SPLINE
SPL {X  -159.990, Y  +457.098, Z    +0.000, E1   +61.912, E3 +184875.364}
SPL {X  -159.990, Y  +442.075, Z    +0.000, E1   +62.596, E3 +184887.140}
SPL {X  -159.990, Y  +430.868, Z    +0.000, E1   +63.135, E3 +184895.393}
SPL {X  -159.990, Y  +416.857, Z    +0.000, E1   +63.835, E3 +184905.060}
SPL {X  -159.990, Y  +402.942, Z    +0.000, E1   +64.377, E3 +184915.289}
SPL {X  -159.990, Y  +382.745, Z    +0.000, E1   +65.209, E3 +184929.203}
SPL {X  -158.929, Y  +364.101, Z    +0.000, E1   +65.981, E3 +184940.958}
SPL {X  -156.693, Y  +350.188, Z    +0.000, E1   +66.345, E3 +184951.082}
SPL {X  -154.578, Y  +341.238, Z    +0.000, E1   +66.113, E3 +184960.840}
SPL {X  -151.958, Y  +332.444, Z    +0.000, E1   +65.791, E3 +184971.400}
SPL {X  -148.012, Y  +321.760, Z    +0.000, E1   +65.212, E3 +184985.033}
SPL {X  -145.172, Y  +315.256, Z    +0.000, E1   +64.753, E3 +184993.738}
SPL {X  -142.205, Y  +309.188, Z    +0.000, E1   +64.322, E3 +185001.991}
SPL {X  -138.693, Y  +302.744, Z    +0.000, E1   +63.741, E3 +185011.048}
SPL {X  -135.977, Y  +298.197, Z    +0.000, E1   +63.280, E3 +185017.568}
SPL {X  -132.828, Y  +293.318, Z    +0.000, E1   +62.759, E3 +185024.622}
SPL {X  -129.451, Y  +288.482, Z    +0.000, E1   +62.137, E3 +185031.725}
SPL {X  -102.192, Y  +259.400, Z    +0.000, E1   +52.167, E3 +185148.272}
ENDSPLINE

SPLINE
SPL {X  -140.725, Y  +306.386, Z    +0.000, E1   +41.058, E3 +185273.166}
SPL {X  -153.851, Y  +338.606, Z    +0.000, E1   +29.149, E3 +185289.783}
SPL {X  -158.264, Y  +359.064, Z    +0.000, E1   +18.155, E3 +185294.734}
SPL {X  -159.641, Y  +371.933, Z    +0.000, E1    +9.693, E3 +185296.470}
SPL {X  -159.986, Y  +381.420, Z    +0.000, E1    +2.704, E3 +185297.035}
SPL {X  -159.990, Y  +384.527, Z    +0.000, E1    -0.013, E3 +185297.095}
SPL {X  -159.990, Y  +385.909, Z    +0.000, E1    -1.800, E3 +185297.113}
SPL {X  -159.990, Y  +389.230, Z    +0.000, E1    -6.815, E3 +185297.237}
SPL {X  -159.990, Y  +395.332, Z    +0.000, E1   -17.451, E3 +185297.720}
SPL {X  -159.990, Y  +403.857, Z    +0.000, E1   -31.979, E3 +185298.945}
SPL {X  -159.990, Y  +417.858, Z    +0.000, E1   -47.695, E3 +185302.430}
SPL {X  -159.990, Y  +475.808, Z    +0.000, E1   -64.751, E3 +185326.384}
SPL {X  -159.990, Y  +590.266, Z    +0.000, E1   -66.680, E3 +185409.501}
SPL {X  -159.990, Y  +605.903, Z    +0.000, E1   -66.635, E3 +185423.920}
SPL {X  -159.990, Y  +620.525, Z    +0.000, E1   -66.669, E3 +185437.254}
SPL {X  -159.990, Y  +638.202, Z    +0.000, E1   -66.649, E3 +185453.504}
SPL {X  -159.990, Y  +654.774, Z    +0.000, E1   -66.658, E3 +185468.673}
SPL {X  -159.990, Y  +671.049, Z    +0.000, E1   -66.648, E3 +185483.604}
SPL {X  -159.584, Y  +682.893, Z    +0.000, E1   -66.583, E3 +185494.902}
SPL {X  -158.845, Y  +690.607, Z    +0.000, E1   -66.486, E3 +185502.754}
SPL {X  -157.279, Y  +700.830, Z    +0.000, E1   -66.296, E3 +185513.735}
SPL {X  -154.589, Y  +712.719, Z    +0.000, E1   -65.941, E3 +185527.378}
SPL {X  -151.974, Y  +721.507, Z    +0.000, E1   -65.548, E3 +185538.131}
SPL {X  -149.510, Y  +728.452, Z    +0.000, E1   -65.197, E3 +185546.973}
SPL {X  -146.809, Y  +735.092, Z    +0.000, E1   -64.789, E3 +185555.720}
SPL {X  -143.550, Y  +742.141, Z    +0.000, E1   -64.312, E3 +185565.239}
SPL {X  -140.309, Y  +748.378, Z    +0.000, E1   -63.779, E3 +185573.972}
SPL {X  -136.621, Y  +754.755, Z    +0.000, E1   -63.190, E3 +185583.089}
SPL {X  -133.172, Y  +760.168, Z    +0.000, E1   -62.565, E3 +185591.010}
SPL {X  -130.070, Y  +764.659, Z    +0.000, E1   -62.024, E3 +185597.606}
SPL {X  -103.420, Y  +793.570, Z    +0.000, E1   -51.337, E3 +185727.505}
ENDSPLINE

SPLINE
SPL {X  -141.359, Y  +746.429, Z    +0.000, E1   -41.207, E3 +185845.719}
SPL {X  -153.791, Y  +715.605, Z    +0.000, E1   -29.700, E3 +185860.488}
SPL {X  -157.923, Y  +697.131, Z    +0.000, E1   -19.758, E3 +185865.020}
SPL {X  -159.426, Y  +684.927, Z    +0.000, E1   -11.876, E3 +185866.749}
SPL {X  -159.929, Y  +675.915, Z    +0.000, E1    -5.290, E3 +185867.459}
SPL {X  -159.990, Y  +669.794, Z    +0.000, E1    -0.371, E3 +185867.633}
SPL {X  -159.990, Y  +668.338, Z    +0.000, E1    +1.468, E3 +185867.649}
SPL {X  -159.990, Y  +664.217, Z    +0.000, E1    +7.944, E3 +185867.802}
SPL {X  -159.990, Y  +657.963, Z    +0.000, E1   +19.417, E3 +185868.298}
SPL {X  -159.990, Y  +649.570, Z    +0.000, E1   +33.681, E3 +185869.522}
SPL {X  -159.990, Y  +636.314, Z    +0.000, E1   +48.490, E3 +185872.825}
SPL {X  -159.990, Y  +588.081, Z    +0.000, E1   +63.406, E3 +185894.007}
SPL {X  -159.990, Y  +471.514, Z    +0.000, E1   +66.231, E3 +185977.515}
SPL {X  -159.990, Y  +458.012, Z    +0.000, E1   +66.224, E3 +185990.144}
SPL {X  -159.990, Y  +445.900, Z    +0.000, E1   +66.225, E3 +186001.458}
ENDSPLINE

SPLINE
SPL {X  -159.990, Y  +465.730, Z    +0.000, E1   +61.693, E3 +186015.282}
ENDSPLINE

SPLINE
SPL {X  -159.990, Y  +446.910, Z    +0.000, E1   +62.394, E3 +186031.502}
SPL {X  -159.990, Y  +430.868, Z    +0.000, E1   +63.135, E3 +186043.542}
SPL {X  -159.990, Y  +416.857, Z    +0.000, E1   +63.835, E3 +186053.208}
SPL {X  -159.990, Y  +402.942, Z    +0.000, E1   +64.377, E3 +186063.437}
SPL {X  -159.990, Y  +382.745, Z    +0.000, E1   +65.209, E3 +186077.352}
SPL {X  -158.342, Y  +359.598, Z    +0.000, E1   +66.150, E3 +186092.056}
SPL {X  -155.453, Y  +344.669, Z    +0.000, E1   +66.270, E3 +186104.898}
SPL {X  -151.958, Y  +332.444, Z    +0.000, E1   +65.791, E3 +186119.548}
SPL {X  -148.012, Y  +321.760, Z    +0.000, E1   +65.212, E3 +186133.181}
SPL {X  -144.181, Y  +313.155, Z    +0.000, E1   +64.628, E3 +186144.691}
SPL {X  -141.300, Y  +307.460, Z    +0.000, E1   +64.150, E3 +186152.583}
SPL {X  -138.693, Y  +302.744, Z    +0.000, E1   +63.741, E3 +186159.196}
SPL {X  -135.031, Y  +296.690, Z    +0.000, E1   +63.147, E3 +186167.858}
SPL {X  -130.494, Y  +289.936, Z    +0.000, E1   +62.364, E3 +186177.696}
SPL {X  -102.192, Y  +259.400, Z    +0.000, E1   +52.167, E3 +186296.420}
ENDSPLINE

SPLINE
SPL {X  -140.725, Y  +306.386, Z    +0.000, E1   +41.058, E3 +186421.314}
SPL {X  -153.851, Y  +338.606, Z    +0.000, E1   +29.149, E3 +186437.932}
SPL {X  -158.264, Y  +359.064, Z    +0.000, E1   +18.155, E3 +186442.883}
SPL {X  -159.641, Y  +371.933, Z    +0.000, E1    +9.693, E3 +186444.618}
SPL {X  -159.986, Y  +381.420, Z    +0.000, E1    +2.704, E3 +186445.183}
SPL {X  -159.990, Y  +384.527, Z    +0.000, E1    -0.013, E3 +186445.244}
SPL {X  -159.990, Y  +386.984, Z    +0.000, E1    -3.187, E3 +186445.295}
SPL {X  -159.990, Y  +392.544, Z    +0.000, E1   -12.471, E3 +186445.608}
SPL {X  -159.990, Y  +397.827, Z    +0.000, E1   -22.184, E3 +186446.129}
SPL {X  -159.990, Y  +403.857, Z    +0.000, E1   -31.979, E3 +186447.093}
SPL {X  -159.990, Y  +417.858, Z    +0.000, E1   -47.695, E3 +186450.579}
SPL {X  -159.990, Y  +475.808, Z    +0.000, E1   -64.751, E3 +186474.532}
SPL {X  -159.990, Y  +586.159, Z    +0.000, E1   -66.648, E3 +186553.948}
SPL {X  -159.990, Y  +602.026, Z    +0.000, E1   -66.659, E3 +186568.465}
SPL {X  -159.990, Y  +620.525, Z    +0.000, E1   -66.669, E3 +186585.402}
SPL {X  -159.990, Y  +638.202, Z    +0.000, E1   -66.649, E3 +186601.652}
SPL {X  -159.990, Y  +654.774, Z    +0.000, E1   -66.658, E3 +186616.821}
SPL {X  -159.990, Y  +671.049, Z    +0.000, E1   -66.648, E3 +186631.752}
SPL {X  -159.230, Y  +687.071, Z    +0.000, E1   -66.569, E3 +186647.193}
SPL {X  -157.279, Y  +700.830, Z    +0.000, E1   -66.296, E3 +186661.883}
SPL {X  -154.589, Y  +712.719, Z    +0.000, E1   -65.941, E3 +186675.526}
SPL {X  -151.974, Y  +721.507, Z    +0.000, E1   -65.548, E3 +186686.279}
SPL {X  -149.510, Y  +728.452, Z    +0.000, E1   -65.197, E3 +186695.121}
SPL {X  -145.784, Y  +737.407, Z    +0.000, E1   -64.671, E3 +186706.912}
SPL {X  -141.166, Y  +746.792, Z    +0.000, E1   -63.950, E3 +186719.841}
SPL {X  -136.621, Y  +754.755, Z    +0.000, E1   -63.190, E3 +186731.237}
SPL {X  -133.172, Y  +760.168, Z    +0.000, E1   -62.565, E3 +186739.158}
SPL {X  -130.070, Y  +764.659, Z    +0.000, E1   -62.024, E3 +186745.754}
SPL {X  -103.420, Y  +793.570, Z    +0.000, E1   -51.337, E3 +186875.653}
ENDSPLINE

SPLINE
SPL {X  -132.256, Y  +761.529, Z    +0.000, E1   -44.935, E3 +186981.743}
SPL {X  -148.790, Y  +730.309, Z    +0.000, E1   -35.907, E3 +187003.017}
SPL {X  -157.132, Y  +701.603, Z    +0.000, E1   -22.438, E3 +187012.278}
SPL {X  -159.426, Y  +684.927, Z    +0.000, E1   -11.876, E3 +187014.897}
SPL {X  -159.929, Y  +675.915, Z    +0.000, E1    -5.290, E3 +187015.607}
SPL {X  -159.990, Y  +669.794, Z    +0.000, E1    -0.371, E3 +187015.781}
SPL {X  -159.990, Y  +668.338, Z    +0.000, E1    +1.468, E3 +187015.797}
SPL {X  -159.990, Y  +664.217, Z    +0.000, E1    +7.944, E3 +187015.950}
SPL {X  -159.990, Y  +657.963, Z    +0.000, E1   +19.417, E3 +187016.446}
SPL {X  -159.990, Y  +649.570, Z    +0.000, E1   +33.681, E3 +187017.670}
SPL {X  -159.990, Y  +636.314, Z    +0.000, E1   +48.490, E3 +187020.974}
SPL {X  -159.990, Y  +588.081, Z    +0.000, E1   +63.406, E3 +187042.155}
SPL {X  -159.990, Y  +471.514, Z    +0.000, E1   +66.231, E3 +187125.663}
SPL {X  -159.990, Y  +458.012, Z    +0.000, E1   +66.224, E3 +187138.293}
SPL {X  -159.990, Y  +445.900, Z    +0.000, E1   +66.225, E3 +187149.606}
ENDSPLINE

SPLINE
SPL {X  -159.990, Y  +465.730, Z    +0.000, E1   +61.693, E3 +187163.430}
ENDSPLINE

SPLINE
SPL {X  -159.990, Y  +452.456, Z    +0.000, E1   +62.114, E3 +187175.358}
SPL {X  -159.990, Y  +436.367, Z    +0.000, E1   +62.893, E3 +187187.618}
SPL {X  -159.990, Y  +416.857, Z    +0.000, E1   +63.835, E3 +187201.357}
SPL {X  -159.990, Y  +402.942, Z    +0.000, E1   +64.377, E3 +187211.585}
SPL {X  -159.990, Y  +382.745, Z    +0.000, E1   +65.209, E3 +187225.500}
SPL {X  -158.342, Y  +359.598, Z    +0.000, E1   +66.150, E3 +187240.204}
SPL {X  -155.453, Y  +344.669, Z    +0.000, E1   +66.270, E3 +187253.046}
SPL {X  -151.958, Y  +332.444, Z    +0.000, E1   +65.791, E3 +187267.696}
SPL {X  -148.012, Y  +321.760, Z    +0.000, E1   +65.212, E3 +187281.329}
SPL {X  -144.181, Y  +313.155, Z    +0.000, E1   +64.628, E3 +187292.839}
SPL {X  -141.300, Y  +307.460, Z    +0.000, E1   +64.150, E3 +187300.731}
SPL {X  -138.693, Y  +302.744, Z    +0.000, E1   +63.741, E3 +187307.345}
SPL {X  -135.031, Y  +296.690, Z    +0.000, E1   +63.147, E3 +187316.006}
SPL {X  -130.494, Y  +289.936, Z    +0.000, E1   +62.364, E3 +187325.844}
SPL {X  -102.192, Y  +259.400, Z    +0.000, E1   +52.167, E3 +187444.569}
ENDSPLINE

SPLINE
SPL {X  -140.725, Y  +306.386, Z    +0.000, E1   +41.058, E3 +187569.463}
SPL {X  -153.851, Y  +338.606, Z    +0.000, E1   +29.149, E3 +187586.080}
SPL {X  -157.523, Y  +354.512, Z    +0.000, E1   +20.811, E3 +187590.206}
SPL {X  -159.458, Y  +369.460, Z    +0.000, E1   +11.469, E3 +187592.495}
SPL {X  -159.986, Y  +381.420, Z    +0.000, E1    +2.704, E3 +187593.331}
SPL {X  -159.990, Y  +385.016, Z    +0.000, E1    -0.442, E3 +187593.398}
SPL {X  -159.990, Y  +389.230, Z    +0.000, E1    -6.815, E3 +187593.534}
SPL {X  -159.990, Y  +395.332, Z    +0.000, E1   -17.451, E3 +187594.016}
SPL {X  -159.990, Y  +403.857, Z    +0.000, E1   -31.979, E3 +187595.241}
SPL {X  -159.990, Y  +416.313, Z    +0.000, E1   -46.481, E3 +187598.234}
SPL {X  -159.990, Y  +425.447, Z    +0.000, E1   -52.896, E3 +187601.143}
SPL {X  -159.990, Y  +475.808, Z    +0.000, E1   -64.751, E3 +187622.680}
SPL {X  -159.990, Y  +586.159, Z    +0.000, E1   -66.648, E3 +187702.096}
SPL {X  -159.990, Y  +602.026, Z    +0.000, E1   -66.659, E3 +187716.613}
SPL {X  -159.990, Y  +615.972, Z    +0.000, E1   -66.639, E3 +187729.441}
SPL {X  -159.990, Y  +629.811, Z    +0.000, E1   -66.653, E3 +187742.093}
SPL {X  -159.990, Y  +646.024, Z    +0.000, E1   -66.650, E3 +187756.970}
SPL {X  -159.990, Y  +658.527, Z    +0.000, E1   -66.634, E3 +187768.451}
SPL {X  -159.990, Y  +671.049, Z    +0.000, E1   -66.648, E3 +187779.900}
SPL {X  -159.584, Y  +682.893, Z    +0.000, E1   -66.583, E3 +187791.198}
SPL {X  -158.332, Y  +694.472, Z    +0.000, E1   -66.450, E3 +187803.071}
SPL {X  -156.148, Y  +706.350, Z    +0.000, E1   -66.133, E3 +187816.283}
SPL {X  -154.052, Y  +714.685, Z    +0.000, E1   -65.842, E3 +187826.070}
SPL {X  -151.381, Y  +723.275, Z    +0.000, E1   -65.482, E3 +187836.617}
SPL {X  -147.622, Y  +733.180, Z    +0.000, E1   -64.943, E3 +187849.421}
SPL {X  -144.546, Y  +740.079, Z    +0.000, E1   -64.439, E3 +187858.749}
SPL {X  -142.587, Y  +744.066, Z    +0.000, E1   -64.133, E3 +187864.243}
SPL {X  -139.326, Y  +750.145, Z    +0.000, E1   -63.650, E3 +187872.736}
SPL {X  -135.791, Y  +756.103, Z    +0.000, E1   -63.018, E3 +187881.381}
SPL {X  -133.172, Y  +760.168, Z    +0.000, E1   -62.565, E3 +187887.306}
SPL {X  -130.070, Y  +764.659, Z    +0.000, E1   -62.024, E3 +187893.902}
SPL {X  -103.420, Y  +793.570, Z    +0.000, E1   -51.337, E3 +188023.802}
ENDSPLINE

SPLINE
SPL {X  -132.256, Y  +761.529, Z    +0.000, E1   -44.935, E3 +188129.891}
SPL {X  -148.790, Y  +730.309, Z    +0.000, E1   -35.907, E3 +188151.165}
SPL {X  -157.132, Y  +701.603, Z    +0.000, E1   -22.438, E3 +188160.426}
SPL {X  -159.426, Y  +684.927, Z    +0.000, E1   -11.876, E3 +188163.045}
SPL {X  -159.929, Y  +675.915, Z    +0.000, E1    -5.290, E3 +188163.755}
SPL {X  -159.990, Y  +669.794, Z    +0.000, E1    -0.371, E3 +188163.929}
SPL {X  -159.990, Y  +668.338, Z    +0.000, E1    +1.468, E3 +188163.945}
SPL {X  -159.990, Y  +665.597, Z    +0.000, E1    +5.793, E3 +188164.024}
SPL {X  -159.990, Y  +662.769, Z    +0.000, E1   +10.720, E3 +188164.175}
SPL {X  -159.990, Y  +657.963, Z    +0.000, E1   +19.417, E3 +188164.595}
SPL {X  -159.990, Y  +649.570, Z    +0.000, E1   +33.681, E3 +188165.819}
SPL {X  -159.990, Y  +636.314, Z    +0.000, E1   +48.490, E3 +188169.122}
SPL {X  -159.990, Y  +588.081, Z    +0.000, E1   +63.406, E3 +188190.303}
SPL {X  -159.990, Y  +471.514, Z    +0.000, E1   +66.231, E3 +188273.811}
SPL {X  -159.990, Y  +458.012, Z    +0.000, E1   +66.224, E3 +188286.441}
SPL {X  -159.990, Y  +445.900, Z    +0.000, E1   +66.225, E3 +188297.754}
ENDSPLINE

SPLINE
SPL {X  -159.990, Y  +465.730, Z    +0.000, E1   +61.693, E3 +188311.579}
ENDSPLINE

SPLINE
SPL {X  -159.990, Y  +446.910, Z    +0.000, E1   +62.394, E3 +188327.798}
SPL {X  -159.990, Y  +430.868, Z    +0.000, E1   +63.135, E3 +188339.838}
SPL {X  -159.990, Y  +416.857, Z    +0.000, E1   +63.835, E3 +188349.505}
SPL {X  -159.990, Y  +397.192, Z    +0.000, E1   +64.622, E3 +188363.798}
SPL {X  -159.570, Y  +370.917, Z    +0.000, E1   +65.713, E3 +188381.155}
SPL {X  -156.693, Y  +350.188, Z    +0.000, E1   +66.345, E3 +188395.527}
SPL {X  -153.533, Y  +337.508, Z    +0.000, E1   +66.008, E3 +188409.659}
SPL {X  -150.132, Y  +327.208, Z    +0.000, E1   +65.515, E3 +188422.445}
SPL {X  -146.325, Y  +317.802, Z    +0.000, E1   +64.967, E3 +188434.700}
SPL {X  -142.205, Y  +309.188, Z    +0.000, E1   +64.322, E3 +188446.436}
SPL {X  -138.693, Y  +302.744, Z    +0.000, E1   +63.741, E3 +188455.493}
SPL {X  -135.031, Y  +296.690, Z    +0.000, E1   +63.147, E3 +188464.154}
SPL {X  -130.494, Y  +289.936, Z    +0.000, E1   +62.364, E3 +188473.992}
SPL {X  -102.192, Y  +259.400, Z    +0.000, E1   +52.167, E3 +188592.717}
ENDSPLINE

SPLINE
SPL {X  -140.725, Y  +306.386, Z    +0.000, E1   +41.058, E3 +188717.611}
SPL {X  -153.851, Y  +338.606, Z    +0.000, E1   +29.149, E3 +188734.228}
SPL {X  -157.523, Y  +354.512, Z    +0.000, E1   +20.811, E3 +188738.354}
SPL {X  -159.458, Y  +369.460, Z    +0.000, E1   +11.469, E3 +188740.644}
SPL {X  -159.986, Y  +381.420, Z    +0.000, E1    +2.704, E3 +188741.479}
SPL {X  -159.990, Y  +385.016, Z    +0.000, E1    -0.442, E3 +188741.546}
SPL {X  -159.990, Y  +389.230, Z    +0.000, E1    -6.815, E3 +188741.682}
SPL {X  -159.990, Y  +393.768, Z    +0.000, E1   -14.836, E3 +188742.000}
SPL {X  -159.990, Y  +397.827, Z    +0.000, E1   -22.184, E3 +188742.426}
SPL {X  -159.990, Y  +403.857, Z    +0.000, E1   -31.979, E3 +188743.390}
SPL {X  -159.990, Y  +417.858, Z    +0.000, E1   -47.695, E3 +188746.875}
SPL {X  -159.990, Y  +475.808, Z    +0.000, E1   -64.751, E3 +188770.828}
SPL {X  -159.990, Y  +590.266, Z    +0.000, E1   -66.680, E3 +188853.946}
SPL {X  -159.990, Y  +605.903, Z    +0.000, E1   -66.635, E3 +188868.365}
SPL {X  -159.990, Y  +620.525, Z    +0.000, E1   -66.669, E3 +188881.699}
SPL {X  -159.990, Y  +638.202, Z    +0.000, E1   -66.649, E3 +188897.948}
SPL {X  -159.990, Y  +649.814, Z    +0.000, E1   -66.629, E3 +188908.636}
SPL {X  -159.990, Y  +658.527, Z    +0.000, E1   -66.634, E3 +188916.599}
SPL {X  -159.990, Y  +671.049, Z    +0.000, E1   -66.648, E3 +188928.048}
SPL {X  -159.584, Y  +682.893, Z    +0.000, E1   -66.583, E3 +188939.346}
SPL {X  -158.332, Y  +694.472, Z    +0.000, E1   -66.450, E3 +188951.220}
SPL {X  -156.148, Y  +706.350, Z    +0.000, E1   -66.133, E3 +188964.431}
SPL {X  -154.052, Y  +714.685, Z    +0.000, E1   -65.842, E3 +188974.218}
SPL {X  -151.974, Y  +721.507, Z    +0.000, E1   -65.548, E3 +188982.575}
SPL {X  -149.510, Y  +728.452, Z    +0.000, E1   -65.197, E3 +188991.418}
SPL {X  -146.809, Y  +735.092, Z    +0.000, E1   -64.789, E3 +189000.165}
SPL {X  -143.550, Y  +742.141, Z    +0.000, E1   -64.312, E3 +189009.683}
SPL {X  -140.309, Y  +748.378, Z    +0.000, E1   -63.779, E3 +189018.416}
SPL {X  -136.621, Y  +754.755, Z    +0.000, E1   -63.190, E3 +189027.533}
SPL {X  -133.172, Y  +760.168, Z    +0.000, E1   -62.565, E3 +189035.454}
SPL {X  -130.070, Y  +764.659, Z    +0.000, E1   -62.024, E3 +189042.050}
SPL {X  -103.420, Y  +793.570, Z    +0.000, E1   -51.337, E3 +189171.950}
ENDSPLINE

SPLINE
SPL {X  -132.256, Y  +761.529, Z    +0.000, E1   -44.935, E3 +189278.039}
SPL {X  -148.790, Y  +730.309, Z    +0.000, E1   -35.907, E3 +189299.313}
SPL {X  -157.132, Y  +701.603, Z    +0.000, E1   -22.438, E3 +189308.574}
SPL {X  -159.426, Y  +684.927, Z    +0.000, E1   -11.876, E3 +189311.193}
SPL {X  -159.929, Y  +675.915, Z    +0.000, E1    -5.290, E3 +189311.903}
SPL {X  -159.990, Y  +669.794, Z    +0.000, E1    -0.371, E3 +189312.077}
SPL {X  -159.990, Y  +668.338, Z    +0.000, E1    +1.468, E3 +189312.094}
SPL {X  -159.990, Y  +664.217, Z    +0.000, E1    +7.944, E3 +189312.246}
SPL {X  -159.990, Y  +658.787, Z    +0.000, E1   +17.995, E3 +189312.651}
SPL {X  -159.990, Y  +653.215, Z    +0.000, E1   +27.908, E3 +189313.343}
SPL {X  -159.990, Y  +646.194, Z    +0.000, E1   +38.517, E3 +189314.632}
SPL {X  -159.990, Y  +636.314, Z    +0.000, E1   +48.490, E3 +189317.270}
SPL {X  -159.990, Y  +588.081, Z    +0.000, E1   +63.406, E3 +189338.451}
SPL {X  -159.990, Y  +471.514, Z    +0.000, E1   +66.231, E3 +189421.959}
SPL {X  -159.990, Y  +458.012, Z    +0.000, E1   +66.224, E3 +189434.589}
SPL {X  -159.990, Y  +445.900, Z    +0.000, E1   +66.225, E3 +189445.902}
ENDSPLINE

SPLINE
SPL {X  -159.990, Y  +465.730, Z    +0.000, E1   +61.693, E3 +189459.727}
ENDSPLINE

SPLINE
SPL {X  -159.990, Y  +452.456, Z    +0.000, E1   +62.114, E3 +189471.654}
SPL {X  -159.990, Y  +436.367, Z    +0.000, E1   +62.893, E3 +189483.914}
SPL {X  -159.990, Y  +416.857, Z    +0.000, E1   +63.835, E3 +189497.653}
SPL {X  -159.990, Y  +397.192, Z    +0.000, E1   +64.622, E3 +189511.946}
SPL {X  -159.902, Y  +377.209, Z    +0.000, E1   +65.412, E3 +189525.510}
SPL {X  -158.342, Y  +359.598, Z    +0.000, E1   +66.150, E3 +189536.501}
SPL {X  -155.453, Y  +344.669, Z    +0.000, E1   +66.270, E3 +189549.343}
SPL {X  -152.827, Y  +335.165, Z    +0.000, E1   +65.880, E3 +189560.700}
SPL {X  -150.132, Y  +327.208, Z    +0.000, E1   +65.515, E3 +189570.593}
SPL {X  -147.311, Y  +320.081, Z    +0.000, E1   +65.083, E3 +189579.874}
SPL {X  -144.181, Y  +313.155, Z    +0.000, E1   +64.628, E3 +189589.135}
SPL {X  -141.300, Y  +307.460, Z    +0.000, E1   +64.150, E3 +189597.027}
SPL {X  -138.693, Y  +302.744, Z    +0.000, E1   +63.741, E3 +189603.641}
SPL {X  -135.977, Y  +298.197, Z    +0.000, E1   +63.280, E3 +189610.161}
SPL {X  -132.828, Y  +293.318, Z    +0.000, E1   +62.759, E3 +189617.214}
SPL {X  -129.451, Y  +288.482, Z    +0.000, E1   +62.137, E3 +189624.318}
SPL {X  -102.192, Y  +259.400, Z    +0.000, E1   +52.167, E3 +189740.865}
ENDSPLINE

SPLINE
SPL {X  -140.725, Y  +306.386, Z    +0.000, E1   +41.058, E3 +189865.759}
SPL {X  -153.851, Y  +338.606, Z    +0.000, E1   +29.149, E3 +189882.376}
SPL {X  -158.264, Y  +359.064, Z    +0.000, E1   +18.155, E3 +189887.327}
SPL {X  -159.641, Y  +371.933, Z    +0.000, E1    +9.693, E3 +189889.062}
SPL {X  -159.986, Y  +381.420, Z    +0.000, E1    +2.704, E3 +189889.627}
SPL {X  -159.990, Y  +384.527, Z    +0.000, E1    -0.013, E3 +189889.688}
SPL {X  -159.990, Y  +385.909, Z    +0.000, E1    -1.800, E3 +189889.705}
SPL {X  -159.990, Y  +389.230, Z    +0.000, E1    -6.815, E3 +189889.830}
SPL {X  -159.990, Y  +395.332, Z    +0.000, E1   -17.451, E3 +189890.312}
SPL {X  -159.990, Y  +403.857, Z    +0.000, E1   -31.979, E3 +189891.538}
SPL {X  -159.990, Y  +417.858, Z    +0.000, E1   -47.695, E3 +189895.023}
SPL {X  -159.990, Y  +475.808, Z    +0.000, E1   -64.751, E3 +189918.977}
SPL {X  -159.990, Y  +586.159, Z    +0.000, E1   -66.648, E3 +189998.393}
SPL {X  -159.990, Y  +602.026, Z    +0.000, E1   -66.659, E3 +190012.909}
SPL {X  -159.990, Y  +620.525, Z    +0.000, E1   -66.669, E3 +190029.847}
SPL {X  -159.990, Y  +638.202, Z    +0.000, E1   -66.649, E3 +190046.096}
SPL {X  -159.990, Y  +654.774, Z    +0.000, E1   -66.658, E3 +190061.266}
SPL {X  -159.990, Y  +671.049, Z    +0.000, E1   -66.648, E3 +190076.196}
SPL {X  -159.230, Y  +687.071, Z    +0.000, E1   -66.569, E3 +190091.638}
SPL {X  -157.279, Y  +700.830, Z    +0.000, E1   -66.296, E3 +190106.328}
SPL {X  -154.589, Y  +712.719, Z    +0.000, E1   -65.941, E3 +190119.971}
SPL {X  -151.381, Y  +723.275, Z    +0.000, E1   -65.482, E3 +190132.914}
SPL {X  -147.622, Y  +733.180, Z    +0.000, E1   -64.943, E3 +190145.717}
SPL {X  -143.550, Y  +742.141, Z    +0.000, E1   -64.312, E3 +190157.831}
SPL {X  -139.326, Y  +750.145, Z    +0.000, E1   -63.650, E3 +190169.032}
SPL {X  -135.791, Y  +756.103, Z    +0.000, E1   -63.018, E3 +190177.678}
SPL {X  -133.172, Y  +760.168, Z    +0.000, E1   -62.565, E3 +190183.603}
SPL {X  -130.070, Y  +764.659, Z    +0.000, E1   -62.024, E3 +190190.198}
SPL {X  -103.420, Y  +793.570, Z    +0.000, E1   -51.337, E3 +190320.098}
ENDSPLINE

SPLINE
SPL {X  -141.359, Y  +746.429, Z    +0.000, E1   -41.207, E3 +190438.312}
SPL {X  -153.791, Y  +715.605, Z    +0.000, E1   -29.700, E3 +190453.081}
SPL {X  -157.923, Y  +697.131, Z    +0.000, E1   -19.758, E3 +190457.612}
SPL {X  -159.426, Y  +684.927, Z    +0.000, E1   -11.876, E3 +190459.341}
SPL {X  -159.972, Y  +673.894, Z    +0.000, E1    -3.783, E3 +190460.129}
SPL {X  -159.990, Y  +669.020, Z    +0.000, E1    +0.387, E3 +190460.234}
SPL {X  -159.990, Y  +664.217, Z    +0.000, E1    +7.944, E3 +190460.394}
SPL {X  -159.990, Y  +657.963, Z    +0.000, E1   +19.417, E3 +190460.891}
SPL {X  -159.990, Y  +649.570, Z    +0.000, E1   +33.681, E3 +190462.115}
SPL {X  -159.990, Y  +636.314, Z    +0.000, E1   +48.490, E3 +190465.418}
SPL {X  -159.990, Y  +588.081, Z    +0.000, E1   +63.406, E3 +190486.599}
SPL {X  -159.990, Y  +471.514, Z    +0.000, E1   +66.231, E3 +190570.107}
SPL {X  -159.990, Y  +458.012, Z    +0.000, E1   +66.224, E3 +190582.737}
SPL {X  -159.990, Y  +445.900, Z    +0.000, E1   +66.225, E3 +190594.050}
ENDSPLINE

SPLINE
SPL {X  -159.990, Y  +468.953, Z    +0.000, E1   +61.697, E3 +190604.009}
ENDSPLINE

SPLINE
SPL {X  -159.990, Y  +457.098, Z    +0.000, E1   +61.912, E3 +190616.105}
SPL {X  -159.990, Y  +442.075, Z    +0.000, E1   +62.596, E3 +190627.880}
SPL {X  -159.990, Y  +430.868, Z    +0.000, E1   +63.135, E3 +190636.134}
SPL {X  -159.990, Y  +416.857, Z    +0.000, E1   +63.835, E3 +190645.801}
SPL {X  -159.990, Y  +402.942, Z    +0.000, E1   +64.377, E3 +190656.030}
SPL {X  -159.990, Y  +382.745, Z    +0.000, E1   +65.209, E3 +190669.944}
SPL {X  -158.929, Y  +364.101, Z    +0.000, E1   +65.981, E3 +190681.699}
SPL {X  -156.693, Y  +350.188, Z    +0.000, E1   +66.345, E3 +190691.823}
SPL {X  -154.578, Y  +341.238, Z    +0.000, E1   +66.113, E3 +190701.581}
SPL {X  -152.827, Y  +335.165, Z    +0.000, E1   +65.880, E3 +190708.849}
SPL {X  -150.132, Y  +327.208, Z    +0.000, E1   +65.515, E3 +190718.741}
SPL {X  -147.311, Y  +320.081, Z    +0.000, E1   +65.083, E3 +190728.022}
SPL {X  -144.181, Y  +313.155, Z    +0.000, E1   +64.628, E3 +190737.283}
SPL {X  -141.300, Y  +307.460, Z    +0.000, E1   +64.150, E3 +190745.175}
SPL {X  -138.693, Y  +302.744, Z    +0.000, E1   +63.741, E3 +190751.789}
SPL {X  -135.977, Y  +298.197, Z    +0.000, E1   +63.280, E3 +190758.309}
SPL {X  -132.828, Y  +293.318, Z    +0.000, E1   +62.759, E3 +190765.362}
SPL {X  -129.451, Y  +288.482, Z    +0.000, E1   +62.137, E3 +190772.466}
SPL {X  -102.192, Y  +259.400, Z    +0.000, E1   +52.167, E3 +190889.013}
ENDSPLINE

SPLINE
SPL {X  -132.063, Y  +292.188, Z    +0.000, E1   +44.502, E3 +191001.173}
SPL {X  -144.900, Y  +314.671, Z    +0.000, E1   +38.548, E3 +191019.789}
SPL {X  -153.851, Y  +338.606, Z    +0.000, E1   +29.149, E3 +191030.524}
SPL {X  -158.264, Y  +359.064, Z    +0.000, E1   +18.155, E3 +191035.475}
SPL {X  -159.641, Y  +371.933, Z    +0.000, E1    +9.693, E3 +191037.210}
SPL {X  -159.986, Y  +381.420, Z    +0.000, E1    +2.704, E3 +191037.775}
SPL {X  -159.990, Y  +385.016, Z    +0.000, E1    -0.442, E3 +191037.842}
SPL {X  -159.990, Y  +389.230, Z    +0.000, E1    -6.815, E3 +191037.978}
SPL {X  -159.990, Y  +395.332, Z    +0.000, E1   -17.451, E3 +191038.461}
SPL {X  -159.990, Y  +403.857, Z    +0.000, E1   -31.979, E3 +191039.686}
SPL {X  -159.990, Y  +416.313, Z    +0.000, E1   -46.481, E3 +191042.678}
SPL {X  -159.990, Y  +425.447, Z    +0.000, E1   -52.896, E3 +191045.587}
SPL {X  -159.990, Y  +475.808, Z    +0.000, E1   -64.751, E3 +191067.125}
SPL {X  -159.990, Y  +590.266, Z    +0.000, E1   -66.680, E3 +191150.242}
SPL {X  -159.990, Y  +611.678, Z    +0.000, E1   -66.672, E3 +191169.882}
SPL {X  -159.990, Y  +629.811, Z    +0.000, E1   -66.653, E3 +191186.538}
SPL {X  -159.990, Y  +646.024, Z    +0.000, E1   -66.650, E3 +191201.414}
SPL {X  -159.990, Y  +658.527, Z    +0.000, E1   -66.634, E3 +191212.895}
SPL {X  -159.990, Y  +671.049, Z    +0.000, E1   -66.648, E3 +191224.344}
SPL {X  -159.584, Y  +682.893, Z    +0.000, E1   -66.583, E3 +191235.642}
SPL {X  -158.332, Y  +694.472, Z    +0.000, E1   -66.450, E3 +191247.516}
SPL {X  -156.148, Y  +706.350, Z    +0.000, E1   -66.133, E3 +191260.727}
SPL {X  -154.052, Y  +714.685, Z    +0.000, E1   -65.842, E3 +191270.514}
SPL {X  -151.974, Y  +721.507, Z    +0.000, E1   -65.548, E3 +191278.871}
SPL {X  -149.510, Y  +728.452, Z    +0.000, E1   -65.197, E3 +191287.714}
SPL {X  -145.784, Y  +737.407, Z    +0.000, E1   -64.671, E3 +191299.505}
SPL {X  -141.166, Y  +746.792, Z    +0.000, E1   -63.950, E3 +191312.434}
SPL {X  -136.621, Y  +754.755, Z    +0.000, E1   -63.190, E3 +191323.829}
SPL {X  -133.172, Y  +760.168, Z    +0.000, E1   -62.565, E3 +191331.751}
SPL {X  -130.070, Y  +764.659, Z    +0.000, E1   -62.024, E3 +191338.346}
SPL {X  -103.420, Y  +793.570, Z    +0.000, E1   -51.337, E3 +191468.246}
ENDSPLINE

SPLINE
SPL {X  -132.256, Y  +761.529, Z    +0.000, E1   -44.935, E3 +191574.336}
SPL {X  -148.790, Y  +730.309, Z    +0.000, E1   -35.907, E3 +191595.609}
SPL {X  -155.396, Y  +709.563, Z    +0.000, E1   -26.693, E3 +191603.111}
SPL {X  -157.923, Y  +697.131, Z    +0.000, E1   -19.758, E3 +191605.760}
SPL {X  -159.426, Y  +684.927, Z    +0.000, E1   -11.876, E3 +191607.489}
SPL {X  -159.972, Y  +673.894, Z    +0.000, E1    -3.783, E3 +191608.277}
SPL {X  -159.990, Y  +669.561, Z    +0.000, E1    -0.077, E3 +191608.376}
SPL {X  -159.990, Y  +668.338, Z    +0.000, E1    +1.468, E3 +191608.390}
SPL {X  -159.990, Y  +664.217, Z    +0.000, E1    +7.944, E3 +191608.542}
SPL {X  -159.990, Y  +658.787, Z    +0.000, E1   +17.995, E3 +191608.948}
SPL {X  -159.990, Y  +653.215, Z    +0.000, E1   +27.908, E3 +191609.640}
SPL {X  -159.990, Y  +646.194, Z    +0.000, E1   +38.517, E3 +191610.928}
SPL {X  -159.990, Y  +636.314, Z    +0.000, E1   +48.490, E3 +191613.566}
SPL {X  -159.990, Y  +588.081, Z    +0.000, E1   +63.406, E3 +191634.748}
SPL {X  -159.990, Y  +471.514, Z    +0.000, E1   +66.231, E3 +191718.256}
SPL {X  -159.990, Y  +458.012, Z    +0.000, E1   +66.224, E3 +191730.885}
SPL {X  -159.990, Y  +445.900, Z    +0.000, E1   +66.225, E3 +191742.198}
ENDSPLINE

SPLINE
SPL {X  -159.990, Y  +465.730, Z    +0.000, E1   +61.693, E3 +191756.023}
ENDSPLINE

SPLINE
SPL {X  -159.990, Y  +452.456, Z    +0.000, E1   +62.114, E3 +191767.950}
SPL {X  -159.990, Y  +436.367, Z    +0.000, E1   +62.893, E3 +191780.210}
SPL {X  -159.990, Y  +416.857, Z    +0.000, E1   +63.835, E3 +191793.949}
SPL {X  -159.990, Y  +402.942, Z    +0.000, E1   +64.377, E3 +191804.178}
SPL {X  -159.990, Y  +382.745, Z    +0.000, E1   +65.209, E3 +191818.092}
SPL {X  -158.929, Y  +364.101, Z    +0.000, E1   +65.981, E3 +191829.847}
SPL {X  -156.693, Y  +350.188, Z    +0.000, E1   +66.345, E3 +191839.971}
SPL {X  -154.578, Y  +341.238, Z    +0.000, E1   +66.113, E3 +191849.729}
SPL {X  -151.958, Y  +332.444, Z    +0.000, E1   +65.791, E3 +191860.289}
SPL {X  -148.012, Y  +321.760, Z    +0.000, E1   +65.212, E3 +191873.922}
SPL {X  -144.181, Y  +313.155, Z    +0.000, E1   +64.628, E3 +191885.432}
SPL {X  -141.300, Y  +307.460, Z    +0.000, E1   +64.150, E3 +191893.323}
SPL {X  -138.693, Y  +302.744, Z    +0.000, E1   +63.741, E3 +191899.937}
SPL {X  -135.977, Y  +298.197, Z    +0.000, E1   +63.280, E3 +191906.457}
SPL {X  -132.828, Y  +293.318, Z    +0.000, E1   +62.759, E3 +191913.511}
SPL {X  -129.451, Y  +288.482, Z    +0.000, E1   +62.137, E3 +191920.614}
SPL {X  -102.192, Y  +259.400, Z    +0.000, E1   +52.167, E3 +192037.161}
ENDSPLINE

SPLINE
SPL {X  -140.725, Y  +306.386, Z    +0.000, E1   +41.058, E3 +192162.055}
SPL {X  -153.851, Y  +338.606, Z    +0.000, E1   +29.149, E3 +192178.672}
SPL {X  -158.264, Y  +359.064, Z    +0.000, E1   +18.155, E3 +192183.623}
SPL {X  -159.641, Y  +371.933, Z    +0.000, E1    +9.693, E3 +192185.359}
SPL {X  -159.986, Y  +381.420, Z    +0.000, E1    +2.704, E3 +192185.924}
SPL {X  -159.990, Y  +385.016, Z    +0.000, E1    -0.442, E3 +192185.990}
SPL {X  -159.990, Y  +389.230, Z    +0.000, E1    -6.815, E3 +192186.126}
SPL {X  -159.990, Y  +395.332, Z    +0.000, E1   -17.451, E3 +192186.609}
SPL {X  -159.990, Y  +403.857, Z    +0.000, E1   -31.979, E3 +192187.834}
SPL {X  -159.990, Y  +416.313, Z    +0.000, E1   -46.481, E3 +192190.826}
SPL {X  -159.990, Y  +425.447, Z    +0.000, E1   -52.896, E3 +192193.735}
SPL {X  -159.990, Y  +475.808, Z    +0.000, E1   -64.751, E3 +192215.273}
SPL {X  -159.990, Y  +590.266, Z    +0.000, E1   -66.680, E3 +192298.390}
SPL {X  -159.990, Y  +611.678, Z    +0.000, E1   -66.672, E3 +192318.030}
SPL {X  -159.990, Y  +625.813, Z    +0.000, E1   -66.632, E3 +192331.061}
SPL {X  -159.990, Y  +638.202, Z    +0.000, E1   -66.649, E3 +192342.393}
SPL {X  -159.990, Y  +654.774, Z    +0.000, E1   -66.658, E3 +192357.562}
SPL {X  -159.990, Y  +671.049, Z    +0.000, E1   -66.648, E3 +192372.493}
SPL {X  -159.584, Y  +682.893, Z    +0.000, E1   -66.583, E3 +192383.790}
SPL {X  -158.332, Y  +694.472, Z    +0.000, E1   -66.450, E3 +192395.664}
SPL {X  -156.148, Y  +706.350, Z    +0.000, E1   -66.133, E3 +192408.875}
SPL {X  -154.052, Y  +714.685, Z    +0.000, E1   -65.842, E3 +192418.663}
SPL {X  -151.381, Y  +723.275, Z    +0.000, E1   -65.482, E3 +192429.210}
SPL {X  -147.622, Y  +733.180, Z    +0.000, E1   -64.943, E3 +192442.013}
SPL {X  -144.546, Y  +740.079, Z    +0.000, E1   -64.439, E3 +192451.342}
SPL {X  -141.166, Y  +746.792, Z    +0.000, E1   -63.950, E3 +192460.582}
SPL {X  -136.621, Y  +754.755, Z    +0.000, E1   -63.190, E3 +192471.978}
SPL {X  -133.172, Y  +760.168, Z    +0.000, E1   -62.565, E3 +192479.899}
SPL {X  -130.070, Y  +764.659, Z    +0.000, E1   -62.024, E3 +192486.494}
SPL {X  -103.420, Y  +793.570, Z    +0.000, E1   -51.337, E3 +192616.394}
ENDSPLINE

SPLINE
SPL {X  -132.256, Y  +761.529, Z    +0.000, E1   -44.935, E3 +192722.484}
SPL {X  -148.790, Y  +730.309, Z    +0.000, E1   -35.907, E3 +192743.757}
SPL {X  -157.132, Y  +701.603, Z    +0.000, E1   -22.438, E3 +192753.018}
SPL {X  -159.426, Y  +684.927, Z    +0.000, E1   -11.876, E3 +192755.637}
SPL {X  -159.929, Y  +675.915, Z    +0.000, E1    -5.290, E3 +192756.348}
SPL {X  -159.990, Y  +669.794, Z    +0.000, E1    -0.371, E3 +192756.521}
SPL {X  -159.990, Y  +668.338, Z    +0.000, E1    +1.468, E3 +192756.538}
SPL {X  -159.990, Y  +665.597, Z    +0.000, E1    +5.793, E3 +192756.617}
SPL {X  -159.990, Y  +662.769, Z    +0.000, E1   +10.720, E3 +192756.768}
SPL {X  -159.990, Y  +658.787, Z    +0.000, E1   +17.995, E3 +192757.096}
SPL {X  -159.990, Y  +653.215, Z    +0.000, E1   +27.908, E3 +192757.788}
SPL {X  -159.990, Y  +646.194, Z    +0.000, E1   +38.517, E3 +192759.076}
SPL {X  -159.990, Y  +636.314, Z    +0.000, E1   +48.490, E3 +192761.714}
SPL {X  -159.990, Y  +588.081, Z    +0.000, E1   +63.406, E3 +192782.896}
SPL {X  -159.990, Y  +471.514, Z    +0.000, E1   +66.231, E3 +192866.404}
SPL {X  -159.990, Y  +458.012, Z    +0.000, E1   +66.224, E3 +192879.033}
SPL {X  -159.990, Y  +445.900, Z    +0.000, E1   +66.225, E3 +192890.346}
ENDSPLINE

SPLINE
SPL {X  -159.990, Y  +465.730, Z    +0.000, E1   +61.693, E3 +192904.171}
ENDSPLINE

SPLINE
SPL {X  -159.990, Y  +446.910, Z    +0.000, E1   +62.394, E3 +192920.391}
SPL {X  -159.990, Y  +430.868, Z    +0.000, E1   +63.135, E3 +192932.430}
SPL {X  -159.990, Y  +416.857, Z    +0.000, E1   +63.835, E3 +192942.097}
SPL {X  -159.990, Y  +402.942, Z    +0.000, E1   +64.377, E3 +192952.326}
SPL {X  -159.990, Y  +382.745, Z    +0.000, E1   +65.209, E3 +192966.240}
SPL {X  -158.342, Y  +359.598, Z    +0.000, E1   +66.150, E3 +192980.945}
SPL {X  -155.453, Y  +344.669, Z    +0.000, E1   +66.270, E3 +192993.787}
SPL {X  -151.958, Y  +332.444, Z    +0.000, E1   +65.791, E3 +193008.437}
SPL {X  -148.012, Y  +321.760, Z    +0.000, E1   +65.212, E3 +193022.070}
SPL {X  -144.181, Y  +313.155, Z    +0.000, E1   +64.628, E3 +193033.580}
SPL {X  -141.300, Y  +307.460, Z    +0.000, E1   +64.150, E3 +193041.471}
SPL {X  -138.693, Y  +302.744, Z    +0.000, E1   +63.741, E3 +193048.085}
SPL {X  -135.031, Y  +296.690, Z    +0.000, E1   +63.147, E3 +193056.747}
SPL {X  -130.494, Y  +289.936, Z    +0.000, E1   +62.364, E3 +193066.585}
SPL {X  -102.192, Y  +259.400, Z    +0.000, E1   +52.167, E3 +193185.309}
ENDSPLINE

SPLINE
SPL {X  -140.725, Y  +306.386, Z    +0.000, E1   +41.058, E3 +193310.203}
SPL {X  -153.851, Y  +338.606, Z    +0.000, E1   +29.149, E3 +193326.820}
SPL {X  -158.264, Y  +359.064, Z    +0.000, E1   +18.155, E3 +193331.772}
SPL {X  -159.641, Y  +371.933, Z    +0.000, E1    +9.693, E3 +193333.507}
SPL {X  -159.986, Y  +381.420, Z    +0.000, E1    +2.704, E3 +193334.072}
SPL {X  -159.990, Y  +384.527, Z    +0.000, E1    -0.013, E3 +193334.132}
SPL {X  -159.990, Y  +386.984, Z    +0.000, E1    -3.187, E3 +193334.184}
SPL {X  -159.990, Y  +392.544, Z    +0.000, E1   -12.471, E3 +193334.497}
SPL {X  -159.990, Y  +397.827, Z    +0.000, E1   -22.184, E3 +193335.018}
SPL {X  -159.990, Y  +403.857, Z    +0.000, E1   -31.979, E3 +193335.982}
SPL {X  -159.990, Y  +417.858, Z    +0.000, E1   -47.695, E3 +193339.467}
SPL {X  -159.990, Y  +475.808, Z    +0.000, E1   -64.751, E3 +193363.421}
SPL {X  -159.990, Y  +590.266, Z    +0.000, E1   -66.680, E3 +193446.538}
SPL {X  -159.990, Y  +611.678, Z    +0.000, E1   -66.672, E3 +193466.178}
SPL {X  -159.990, Y  +625.813, Z    +0.000, E1   -66.632, E3 +193479.209}
SPL {X  -159.990, Y  +638.202, Z    +0.000, E1   -66.649, E3 +193490.541}
SPL {X  -159.990, Y  +654.774, Z    +0.000, E1   -66.658, E3 +193505.710}
SPL {X  -159.990, Y  +671.049, Z    +0.000, E1   -66.648, E3 +193520.641}
SPL {X  -159.230, Y  +687.071, Z    +0.000, E1   -66.569, E3 +193536.082}
SPL {X  -157.779, Y  +698.005, Z    +0.000, E1   -66.341, E3 +193547.701}
SPL {X  -156.148, Y  +706.350, Z    +0.000, E1   -66.133, E3 +193557.024}
SPL {X  -154.052, Y  +714.685, Z    +0.000, E1   -65.842, E3 +193566.811}
SPL {X  -151.974, Y  +721.507, Z    +0.000, E1   -65.548, E3 +193575.168}
SPL {X  -149.510, Y  +728.452, Z    +0.000, E1   -65.197, E3 +193584.010}
SPL {X  -146.809, Y  +735.092, Z    +0.000, E1   -64.789, E3 +193592.757}
SPL {X  -143.550, Y  +742.141, Z    +0.000, E1   -64.312, E3 +193602.276}
SPL {X  -139.326, Y  +750.145, Z    +0.000, E1   -63.650, E3 +193613.477}
SPL {X  -135.791, Y  +756.103, Z    +0.000, E1   -63.018, E3 +193622.122}
SPL {X  -133.172, Y  +760.168, Z    +0.000, E1   -62.565, E3 +193628.047}
SPL {X  -130.070, Y  +764.659, Z    +0.000, E1   -62.024, E3 +193634.643}
SPL {X  -103.420, Y  +793.570, Z    +0.000, E1   -51.337, E3 +193764.542}
ENDSPLINE

SPLINE
SPL {X  -141.359, Y  +746.429, Z    +0.000, E1   -41.207, E3 +193882.756}
SPL {X  -153.791, Y  +715.605, Z    +0.000, E1   -29.700, E3 +193897.525}
SPL {X  -157.923, Y  +697.131, Z    +0.000, E1   -19.758, E3 +193902.057}
SPL {X  -159.426, Y  +684.927, Z    +0.000, E1   -11.876, E3 +193903.786}
SPL {X  -159.972, Y  +673.894, Z    +0.000, E1    -3.783, E3 +193904.574}
SPL {X  -159.990, Y  +669.561, Z    +0.000, E1    -0.077, E3 +193904.672}
SPL {X  -159.990, Y  +668.338, Z    +0.000, E1    +1.468, E3 +193904.686}
SPL {X  -159.990, Y  +664.217, Z    +0.000, E1    +7.944, E3 +193904.839}
SPL {X  -159.990, Y  +658.787, Z    +0.000, E1   +17.995, E3 +193905.244}
SPL {X  -159.990, Y  +653.215, Z    +0.000, E1   +27.908, E3 +193905.936}
SPL {X  -159.990, Y  +646.194, Z    +0.000, E1   +38.517, E3 +193907.225}
SPL {X  -159.990, Y  +636.314, Z    +0.000, E1   +48.490, E3 +193909.863}
SPL {X  -159.990, Y  +588.081, Z    +0.000, E1   +63.406, E3 +193931.044}
SPL {X  -159.990, Y  +471.514, Z    +0.000, E1   +66.231, E3 +194014.552}
SPL {X  -159.990, Y  +458.012, Z    +0.000, E1   +66.224, E3 +194027.181}
SPL {X  -159.990, Y  +445.900, Z    +0.000, E1   +66.225, E3 +194038.495}
ENDSPLINE

SPLINE
SPL {X  -159.990, Y  +465.730, Z    +0.000, E1   +61.693, E3 +194052.319}
ENDSPLINE

SPLINE
SPL {X  -159.990, Y  +452.456, Z    +0.000, E1   +62.114, E3 +194064.247}
SPL {X  -159.990, Y  +436.367, Z    +0.000, E1   +62.893, E3 +194076.506}
SPL {X  -159.990, Y  +416.857, Z    +0.000, E1   +63.835, E3 +194090.245}
SPL {X  -159.990, Y  +402.942, Z    +0.000, E1   +64.377, E3 +194100.474}
SPL {X  -159.990, Y  +382.745, Z    +0.000, E1   +65.209, E3 +194114.389}
SPL {X  -158.342, Y  +359.598, Z    +0.000, E1   +66.150, E3 +194129.093}
SPL {X  -155.453, Y  +344.669, Z    +0.000, E1   +66.270, E3 +194141.935}
SPL {X  -151.958, Y  +332.444, Z    +0.000, E1   +65.791, E3 +194156.585}
SPL {X  -148.012, Y  +321.760, Z    +0.000, E1   +65.212, E3 +194170.218}
SPL {X  -144.181, Y  +313.155, Z    +0.000, E1   +64.628, E3 +194181.728}
SPL {X  -141.300, Y  +307.460, Z    +0.000, E1   +64.150, E3 +194189.620}
SPL {X  -138.693, Y  +302.744, Z    +0.000, E1   +63.741, E3 +194196.234}
SPL {X  -135.031, Y  +296.690, Z    +0.000, E1   +63.147, E3 +194204.895}
SPL {X  -130.494, Y  +289.936, Z    +0.000, E1   +62.364, E3 +194214.733}
SPL {X  -102.192, Y  +259.400, Z    +0.000, E1   +52.167, E3 +194333.457}
ENDSPLINE

SPLINE
SPL {X  -140.725, Y  +306.386, Z    +0.000, E1   +41.058, E3 +194458.351}
SPL {X  -153.851, Y  +338.606, Z    +0.000, E1   +29.149, E3 +194474.969}
SPL {X  -158.264, Y  +359.064, Z    +0.000, E1   +18.155, E3 +194479.920}
SPL {X  -159.641, Y  +371.933, Z    +0.000, E1    +9.693, E3 +194481.655}
SPL {X  -159.986, Y  +381.420, Z    +0.000, E1    +2.704, E3 +194482.220}
SPL {X  -159.990, Y  +384.527, Z    +0.000, E1    -0.013, E3 +194482.281}
SPL {X  -159.990, Y  +386.984, Z    +0.000, E1    -3.187, E3 +194482.332}
SPL {X  -159.990, Y  +392.544, Z    +0.000, E1   -12.471, E3 +194482.645}
SPL {X  -159.990, Y  +397.827, Z    +0.000, E1   -22.184, E3 +194483.166}
SPL {X  -159.990, Y  +403.857, Z    +0.000, E1   -31.979, E3 +194484.130}
SPL {X  -159.990, Y  +417.858, Z    +0.000, E1   -47.695, E3 +194487.616}
SPL {X  -159.990, Y  +475.808, Z    +0.000, E1   -64.751, E3 +194511.569}
SPL {X  -159.990, Y  +590.266, Z    +0.000, E1   -66.680, E3 +194594.687}
SPL {X  -159.990, Y  +611.678, Z    +0.000, E1   -66.672, E3 +194614.326}
SPL {X  -159.990, Y  +625.813, Z    +0.000, E1   -66.632, E3 +194627.357}
SPL {X  -159.990, Y  +638.202, Z    +0.000, E1   -66.649, E3 +194638.689}
SPL {X  -159.990, Y  +654.774, Z    +0.000, E1   -66.658, E3 +194653.858}
SPL {X  -159.990, Y  +671.049, Z    +0.000, E1   -66.648, E3 +194668.789}
SPL {X  -159.230, Y  +687.071, Z    +0.000, E1   -66.569, E3 +194684.230}
SPL {X  -157.279, Y  +700.830, Z    +0.000, E1   -66.296, E3 +194698.920}
SPL {X  -154.589, Y  +712.719, Z    +0.000, E1   -65.941, E3 +194712.563}
SPL {X  -151.381, Y  +723.275, Z    +0.000, E1   -65.482, E3 +194725.506}
SPL {X  -147.622, Y  +733.180, Z    +0.000, E1   -64.943, E3 +194738.310}
SPL {X  -143.550, Y  +742.141, Z    +0.000, E1   -64.312, E3 +194750.424}
SPL {X  -139.326, Y  +750.145, Z    +0.000, E1   -63.650, E3 +194761.625}
SPL {X  -135.791, Y  +756.103, Z    +0.000, E1   -63.018, E3 +194770.270}
SPL {X  -133.172, Y  +760.168, Z    +0.000, E1   -62.565, E3 +194776.195}
SPL {X  -130.070, Y  +764.659, Z    +0.000, E1   -62.024, E3 +194782.791}
SPL {X  -103.420, Y  +793.570, Z    +0.000, E1   -51.337, E3 +194912.690}
ENDSPLINE

SPLINE
SPL {X  -141.359, Y  +746.429, Z    +0.000, E1   -41.207, E3 +195030.904}
SPL {X  -153.791, Y  +715.605, Z    +0.000, E1   -29.700, E3 +195045.674}
SPL {X  -157.923, Y  +697.131, Z    +0.000, E1   -19.758, E3 +195050.205}
SPL {X  -159.426, Y  +684.927, Z    +0.000, E1   -11.876, E3 +195051.934}
SPL {X  -159.972, Y  +673.894, Z    +0.000, E1    -3.783, E3 +195052.722}
SPL {X  -159.990, Y  +669.561, Z    +0.000, E1    -0.077, E3 +195052.820}
SPL {X  -159.990, Y  +668.338, Z    +0.000, E1    +1.468, E3 +195052.834}
SPL {X  -159.990, Y  +664.217, Z    +0.000, E1    +7.944, E3 +195052.987}
SPL {X  -159.990, Y  +658.787, Z    +0.000, E1   +17.995, E3 +195053.392}
SPL {X  -159.990, Y  +653.215, Z    +0.000, E1   +27.908, E3 +195054.084}
SPL {X  -159.990, Y  +646.194, Z    +0.000, E1   +38.517, E3 +195055.373}
SPL {X  -159.990, Y  +636.314, Z    +0.000, E1   +48.490, E3 +195058.011}
SPL {X  -159.990, Y  +588.081, Z    +0.000, E1   +63.406, E3 +195079.192}
SPL {X  -159.990, Y  +471.514, Z    +0.000, E1   +66.231, E3 +195162.700}
SPL {X  -159.990, Y  +458.012, Z    +0.000, E1   +66.224, E3 +195175.330}
SPL {X  -159.990, Y  +445.900, Z    +0.000, E1   +66.225, E3 +195186.643}
ENDSPLINE

SPLINE
SPL {X  -159.990, Y  +465.730, Z    +0.000, E1   +61.693, E3 +195200.467}
ENDSPLINE

SPLINE
SPL {X  -159.990, Y  +452.456, Z    +0.000, E1   +62.114, E3 +195212.395}
SPL {X  -159.990, Y  +436.367, Z    +0.000, E1   +62.893, E3 +195224.655}
SPL {X  -159.990, Y  +416.857, Z    +0.000, E1   +63.835, E3 +195238.394}
SPL {X  -159.990, Y  +402.942, Z    +0.000, E1   +64.377, E3 +195248.623}
SPL {X  -159.990, Y  +382.745, Z    +0.000, E1   +65.209, E3 +195262.537}
SPL {X  -158.342, Y  +359.598, Z    +0.000, E1   +66.150, E3 +195277.241}
SPL {X  -155.453, Y  +344.669, Z    +0.000, E1   +66.270, E3 +195290.083}
SPL {X  -151.958, Y  +332.444, Z    +0.000, E1   +65.791, E3 +195304.733}
SPL {X  -148.012, Y  +321.760, Z    +0.000, E1   +65.212, E3 +195318.366}
SPL {X  -144.181, Y  +313.155, Z    +0.000, E1   +64.628, E3 +195329.876}
SPL {X  -141.300, Y  +307.460, Z    +0.000, E1   +64.150, E3 +195337.768}
SPL {X  -138.693, Y  +302.744, Z    +0.000, E1   +63.741, E3 +195344.382}
SPL {X  -135.031, Y  +296.690, Z    +0.000, E1   +63.147, E3 +195353.043}
SPL {X  -130.494, Y  +289.936, Z    +0.000, E1   +62.364, E3 +195362.881}
SPL {X  -102.192, Y  +259.400, Z    +0.000, E1   +52.167, E3 +195481.606}
ENDSPLINE

SPLINE
SPL {X  -140.725, Y  +306.386, Z    +0.000, E1   +41.058, E3 +195606.500}
SPL {X  -153.851, Y  +338.606, Z    +0.000, E1   +29.149, E3 +195623.117}
SPL {X  -158.264, Y  +359.064, Z    +0.000, E1   +18.155, E3 +195628.068}
SPL {X  -159.641, Y  +371.933, Z    +0.000, E1    +9.693, E3 +195629.803}
SPL {X  -159.986, Y  +381.420, Z    +0.000, E1    +2.704, E3 +195630.368}
SPL {X  -159.990, Y  +384.527, Z    +0.000, E1    -0.013, E3 +195630.429}
SPL {X  -159.990, Y  +386.984, Z    +0.000, E1    -3.187, E3 +195630.480}
SPL {X  -159.990, Y  +390.572, Z    +0.000, E1    -9.243, E3 +195630.639}
SPL {X  -159.990, Y  +395.332, Z    +0.000, E1   -17.451, E3 +195631.053}
SPL {X  -159.990, Y  +403.857, Z    +0.000, E1   -31.979, E3 +195632.278}
SPL {X  -159.990, Y  +416.313, Z    +0.000, E1   -46.481, E3 +195635.271}
SPL {X  -159.990, Y  +425.447, Z    +0.000, E1   -52.896, E3 +195638.180}
SPL {X  -159.990, Y  +475.808, Z    +0.000, E1   -64.751, E3 +195659.717}
SPL {X  -159.990, Y  +586.159, Z    +0.000, E1   -66.648, E3 +195739.133}
SPL {X  -159.990, Y  +602.026, Z    +0.000, E1   -66.659, E3 +195753.650}
SPL {X  -159.990, Y  +615.972, Z    +0.000, E1   -66.639, E3 +195766.478}
SPL {X  -159.990, Y  +629.811, Z    +0.000, E1   -66.653, E3 +195779.131}
SPL {X  -159.990, Y  +646.024, Z    +0.000, E1   -66.650, E3 +195794.007}
SPL {X  -159.990, Y  +658.527, Z    +0.000, E1   -66.634, E3 +195805.488}
SPL {X  -159.990, Y  +671.049, Z    +0.000, E1   -66.648, E3 +195816.937}
SPL {X  -159.584, Y  +682.893, Z    +0.000, E1   -66.583, E3 +195828.235}
SPL {X  -158.332, Y  +694.472, Z    +0.000, E1   -66.450, E3 +195840.108}
SPL {X  -156.148, Y  +706.350, Z    +0.000, E1   -66.133, E3 +195853.320}
SPL {X  -154.052, Y  +714.685, Z    +0.000, E1   -65.842, E3 +195863.107}
SPL {X  -151.381, Y  +723.275, Z    +0.000, E1   -65.482, E3 +195873.654}
SPL {X  -147.622, Y  +733.180, Z    +0.000, E1   -64.943, E3 +195886.458}
SPL {X  -144.546, Y  +740.079, Z    +0.000, E1   -64.439, E3 +195895.786}
SPL {X  -141.166, Y  +746.792, Z    +0.000, E1   -63.950, E3 +195905.026}
SPL {X  -136.621, Y  +754.755, Z    +0.000, E1   -63.190, E3 +195916.422}
SPL {X  -133.172, Y  +760.168, Z    +0.000, E1   -62.565, E3 +195924.343}
SPL {X  -130.070, Y  +764.659, Z    +0.000, E1   -62.024, E3 +195930.939}
SPL {X  -103.420, Y  +793.570, Z    +0.000, E1   -51.337, E3 +196060.839}
ENDSPLINE

SPLINE
SPL {X  -141.359, Y  +746.429, Z    +0.000, E1   -41.207, E3 +196179.053}
SPL {X  -153.791, Y  +715.605, Z    +0.000, E1   -29.700, E3 +196193.822}
SPL {X  -157.923, Y  +697.131, Z    +0.000, E1   -19.758, E3 +196198.353}
SPL {X  -159.426, Y  +684.927, Z    +0.000, E1   -11.876, E3 +196200.082}
SPL {X  -159.972, Y  +673.894, Z    +0.000, E1    -3.783, E3 +196200.870}
SPL {X  -159.990, Y  +669.020, Z    +0.000, E1    +0.387, E3 +196200.975}
SPL {X  -159.990, Y  +664.217, Z    +0.000, E1    +7.944, E3 +196201.135}
SPL {X  -159.990, Y  +657.963, Z    +0.000, E1   +19.417, E3 +196201.632}
SPL {X  -159.990, Y  +649.570, Z    +0.000, E1   +33.681, E3 +196202.856}
SPL {X  -159.990, Y  +636.314, Z    +0.000, E1   +48.490, E3 +196206.159}
SPL {X  -159.990, Y  +588.081, Z    +0.000, E1   +63.406, E3 +196227.340}
SPL {X  -159.990, Y  +471.514, Z    +0.000, E1   +66.231, E3 +196310.848}
SPL {X  -159.990, Y  +458.012, Z    +0.000, E1   +66.224, E3 +196323.478}
SPL {X  -159.990, Y  +445.900, Z    +0.000, E1   +66.225, E3 +196334.791}
ENDSPLINE

SPLINE
SPL {X  -159.990, Y  +465.730, Z    +0.000, E1   +61.693, E3 +196348.616}
ENDSPLINE

SPLINE
SPL {X  -159.990, Y  +452.456, Z    +0.000, E1   +62.114, E3 +196360.543}
SPL {X  -159.990, Y  +436.367, Z    +0.000, E1   +62.893, E3 +196372.803}
SPL {X  -159.990, Y  +416.857, Z    +0.000, E1   +63.835, E3 +196386.542}
SPL {X  -159.990, Y  +397.192, Z    +0.000, E1   +64.622, E3 +196400.835}
SPL {X  -159.902, Y  +377.209, Z    +0.000, E1   +65.412, E3 +196414.399}
SPL {X  -158.342, Y  +359.598, Z    +0.000, E1   +66.150, E3 +196425.389}
SPL {X  -155.453, Y  +344.669, Z    +0.000, E1   +66.270, E3 +196438.231}
SPL {X  -152.827, Y  +335.165, Z    +0.000, E1   +65.880, E3 +196449.589}
SPL {X  -150.132, Y  +327.208, Z    +0.000, E1   +65.515, E3 +196459.482}
SPL {X  -147.311, Y  +320.081, Z    +0.000, E1   +65.083, E3 +196468.763}
SPL {X  -144.181, Y  +313.155, Z    +0.000, E1   +64.628, E3 +196478.024}
SPL {X  -141.300, Y  +307.460, Z    +0.000, E1   +64.150, E3 +196485.916}
SPL {X  -138.693, Y  +302.744, Z    +0.000, E1   +63.741, E3 +196492.530}
SPL {X  -135.031, Y  +296.690, Z    +0.000, E1   +63.147, E3 +196501.191}
SPL {X  -130.494, Y  +289.936, Z    +0.000, E1   +62.364, E3 +196511.029}
SPL {X  -102.192, Y  +259.400, Z    +0.000, E1   +52.167, E3 +196629.754}
ENDSPLINE

SPLINE
SPL {X  -140.725, Y  +306.386, Z    +0.000, E1   +41.058, E3 +196754.648}
SPL {X  -153.851, Y  +338.606, Z    +0.000, E1   +29.149, E3 +196771.265}
SPL {X  -158.264, Y  +359.064, Z    +0.000, E1   +18.155, E3 +196776.216}
SPL {X  -159.641, Y  +371.933, Z    +0.000, E1    +9.693, E3 +196777.951}
SPL {X  -159.986, Y  +381.420, Z    +0.000, E1    +2.704, E3 +196778.516}
SPL {X  -159.990, Y  +384.527, Z    +0.000, E1    -0.013, E3 +196778.577}
SPL {X  -159.990, Y  +385.909, Z    +0.000, E1    -1.800, E3 +196778.594}
SPL {X  -159.990, Y  +389.230, Z    +0.000, E1    -6.815, E3 +196778.719}
SPL {X  -159.990, Y  +395.332, Z    +0.000, E1   -17.451, E3 +196779.201}
SPL {X  -159.990, Y  +403.857, Z    +0.000, E1   -31.979, E3 +196780.427}
SPL {X  -159.990, Y  +417.858, Z    +0.000, E1   -47.695, E3 +196783.912}
SPL {X  -159.990, Y  +475.808, Z    +0.000, E1   -64.751, E3 +196807.865}
SPL {X  -159.990, Y  +586.159, Z    +0.000, E1   -66.648, E3 +196887.282}
SPL {X  -159.990, Y  +602.026, Z    +0.000, E1   -66.659, E3 +196901.798}
SPL {X  -159.990, Y  +620.525, Z    +0.000, E1   -66.669, E3 +196918.736}
SPL {X  -159.990, Y  +638.202, Z    +0.000, E1   -66.649, E3 +196934.985}
SPL {X  -159.990, Y  +654.774, Z    +0.000, E1   -66.658, E3 +196950.155}
SPL {X  -159.990, Y  +671.049, Z    +0.000, E1   -66.648, E3 +196965.085}
SPL {X  -159.230, Y  +687.071, Z    +0.000, E1   -66.569, E3 +196980.527}
SPL {X  -157.279, Y  +700.830, Z    +0.000, E1   -66.296, E3 +196995.217}
SPL {X  -154.589, Y  +712.719, Z    +0.000, E1   -65.941, E3 +197008.859}
SPL {X  -151.381, Y  +723.275, Z    +0.000, E1   -65.482, E3 +197021.803}
SPL {X  -147.622, Y  +733.180, Z    +0.000, E1   -64.943, E3 +197034.606}
SPL {X  -143.550, Y  +742.141, Z    +0.000, E1   -64.312, E3 +197046.720}
SPL {X  -139.326, Y  +750.145, Z    +0.000, E1   -63.650, E3 +197057.921}
SPL {X  -135.791, Y  +756.103, Z    +0.000, E1   -63.018, E3 +197066.567}
SPL {X  -133.172, Y  +760.168, Z    +0.000, E1   -62.565, E3 +197072.491}
SPL {X  -130.070, Y  +764.659, Z    +0.000, E1   -62.024, E3 +197079.087}
SPL {X  -103.420, Y  +793.570, Z    +0.000, E1   -51.337, E3 +197208.987}
ENDSPLINE

SPLINE
SPL {X  -141.359, Y  +746.429, Z    +0.000, E1   -41.207, E3 +197327.201}
SPL {X  -153.791, Y  +715.605, Z    +0.000, E1   -29.700, E3 +197341.970}
SPL {X  -157.923, Y  +697.131, Z    +0.000, E1   -19.758, E3 +197346.501}
SPL {X  -159.426, Y  +684.927, Z    +0.000, E1   -11.876, E3 +197348.230}
SPL {X  -159.972, Y  +673.894, Z    +0.000, E1    -3.783, E3 +197349.018}
SPL {X  -159.990, Y  +669.561, Z    +0.000, E1    -0.077, E3 +197349.117}
SPL {X  -159.990, Y  +668.338, Z    +0.000, E1    +1.468, E3 +197349.131}
SPL {X  -159.990, Y  +664.217, Z    +0.000, E1    +7.944, E3 +197349.283}
SPL {X  -159.990, Y  +658.787, Z    +0.000, E1   +17.995, E3 +197349.688}
SPL {X  -159.990, Y  +653.215, Z    +0.000, E1   +27.908, E3 +197350.380}
SPL {X  -159.990, Y  +646.194, Z    +0.000, E1   +38.517, E3 +197351.669}
SPL {X  -159.990, Y  +636.314, Z    +0.000, E1   +48.490, E3 +197354.307}
SPL {X  -159.990, Y  +588.081, Z    +0.000, E1   +63.406, E3 +197375.488}
SPL {X  -159.990, Y  +471.514, Z    +0.000, E1   +66.231, E3 +197458.996}
SPL {X  -159.990, Y  +458.012, Z    +0.000, E1   +66.224, E3 +197471.626}
SPL {X  -159.990, Y  +445.900, Z    +0.000, E1   +66.225, E3 +197482.939}
ENDSPLINE

SPLINE
SPL {X  -159.990, Y  +465.730, Z    +0.000, E1   +61.693, E3 +197496.764}
ENDSPLINE

SPLINE
SPL {X  -159.990, Y  +446.910, Z    +0.000, E1   +62.394, E3 +197512.983}
SPL {X  -159.990, Y  +430.868, Z    +0.000, E1   +63.135, E3 +197525.023}
SPL {X  -159.990, Y  +416.857, Z    +0.000, E1   +63.835, E3 +197534.690}
SPL {X  -159.990, Y  +397.192, Z    +0.000, E1   +64.622, E3 +197548.983}
SPL {X  -159.570, Y  +370.917, Z    +0.000, E1   +65.713, E3 +197566.340}
SPL {X  -156.693, Y  +350.188, Z    +0.000, E1   +66.345, E3 +197580.712}
SPL {X  -153.533, Y  +337.508, Z    +0.000, E1   +66.008, E3 +197594.844}
SPL {X  -150.132, Y  +327.208, Z    +0.000, E1   +65.515, E3 +197607.630}
SPL {X  -146.325, Y  +317.802, Z    +0.000, E1   +64.967, E3 +197619.885}
SPL {X  -142.205, Y  +309.188, Z    +0.000, E1   +64.322, E3 +197631.621}
SPL {X  -138.693, Y  +302.744, Z    +0.000, E1   +63.741, E3 +197640.678}
SPL {X  -135.977, Y  +298.197, Z    +0.000, E1   +63.280, E3 +197647.198}
SPL {X  -132.828, Y  +293.318, Z    +0.000, E1   +62.759, E3 +197654.251}
SPL {X  -129.451, Y  +288.482, Z    +0.000, E1   +62.137, E3 +197661.355}
SPL {X  -102.192, Y  +259.400, Z    +0.000, E1   +52.167, E3 +197777.902}
ENDSPLINE

SPLINE
SPL {X  -140.725, Y  +306.386, Z    +0.000, E1   +41.058, E3 +197902.796}
SPL {X  -153.851, Y  +338.606, Z    +0.000, E1   +29.149, E3 +197919.413}
SPL {X  -158.264, Y  +359.064, Z    +0.000, E1   +18.155, E3 +197924.364}
SPL {X  -159.641, Y  +371.933, Z    +0.000, E1    +9.693, E3 +197926.099}
SPL {X  -159.986, Y  +381.420, Z    +0.000, E1    +2.704, E3 +197926.664}
SPL {X  -159.990, Y  +384.527, Z    +0.000, E1    -0.013, E3 +197926.725}
SPL {X  -159.990, Y  +386.984, Z    +0.000, E1    -3.187, E3 +197926.777}
SPL {X  -159.990, Y  +392.544, Z    +0.000, E1   -12.471, E3 +197927.090}
SPL {X  -159.990, Y  +397.827, Z    +0.000, E1   -22.184, E3 +197927.611}
SPL {X  -159.990, Y  +403.857, Z    +0.000, E1   -31.979, E3 +197928.575}
SPL {X  -159.990, Y  +417.858, Z    +0.000, E1   -47.695, E3 +197932.060}
SPL {X  -159.990, Y  +475.808, Z    +0.000, E1   -64.751, E3 +197956.014}
SPL {X  -159.990, Y  +590.266, Z    +0.000, E1   -66.680, E3 +198039.131}
SPL {X  -159.990, Y  +611.678, Z    +0.000, E1   -66.672, E3 +198058.771}
SPL {X  -159.990, Y  +625.813, Z    +0.000, E1   -66.632, E3 +198071.802}
SPL {X  -159.990, Y  +638.202, Z    +0.000, E1   -66.649, E3 +198083.133}
SPL {X  -159.990, Y  +654.774, Z    +0.000, E1   -66.658, E3 +198098.303}
SPL {X  -159.990, Y  +671.049, Z    +0.000, E1   -66.648, E3 +198113.233}
SPL {X  -159.230, Y  +687.071, Z    +0.000, E1   -66.569, E3 +198128.675}
SPL {X  -157.279, Y  +700.830, Z    +0.000, E1   -66.296, E3 +198143.365}
SPL {X  -154.589, Y  +712.719, Z    +0.000, E1   -65.941, E3 +198157.008}
SPL {X  -151.381, Y  +723.275, Z    +0.000, E1   -65.482, E3 +198169.951}
SPL {X  -147.622, Y  +733.180, Z    +0.000, E1   -64.943, E3 +198182.754}
SPL {X  -143.550, Y  +742.141, Z    +0.000, E1   -64.312, E3 +198194.868}
SPL {X  -139.326, Y  +750.145, Z    +0.000, E1   -63.650, E3 +198206.069}
SPL {X  -135.791, Y  +756.103, Z    +0.000, E1   -63.018, E3 +198214.715}
SPL {X  -133.172, Y  +760.168, Z    +0.000, E1   -62.565, E3 +198220.640}
SPL {X  -130.070, Y  +764.659, Z    +0.000, E1   -62.024, E3 +198227.235}
SPL {X  -103.420, Y  +793.570, Z    +0.000, E1   -51.337, E3 +198357.135}
ENDSPLINE

SPLINE
SPL {X  -141.359, Y  +746.429, Z    +0.000, E1   -41.207, E3 +198475.349}
SPL {X  -153.791, Y  +715.605, Z    +0.000, E1   -29.700, E3 +198490.118}
SPL {X  -157.923, Y  +697.131, Z    +0.000, E1   -19.758, E3 +198494.649}
SPL {X  -159.426, Y  +684.927, Z    +0.000, E1   -11.876, E3 +198496.378}
SPL {X  -159.972, Y  +673.894, Z    +0.000, E1    -3.783, E3 +198497.166}
SPL {X  -159.990, Y  +669.561, Z    +0.000, E1    -0.077, E3 +198497.265}
SPL {X  -159.990, Y  +668.338, Z    +0.000, E1    +1.468, E3 +198497.279}
SPL {X  -159.990, Y  +664.217, Z    +0.000, E1    +7.944, E3 +198497.431}
SPL {X  -159.990, Y  +658.787, Z    +0.000, E1   +17.995, E3 +198497.836}
SPL {X  -159.990, Y  +653.215, Z    +0.000, E1   +27.908, E3 +198498.528}
SPL {X  -159.990, Y  +646.194, Z    +0.000, E1   +38.517, E3 +198499.817}
SPL {X  -159.990, Y  +636.314, Z    +0.000, E1   +48.490, E3 +198502.455}
SPL {X  -159.990, Y  +588.081, Z    +0.000, E1   +63.406, E3 +198523.637}
SPL {X  -159.990, Y  +471.514, Z    +0.000, E1   +66.231, E3 +198607.145}
SPL {X  -159.990, Y  +458.012, Z    +0.000, E1   +66.224, E3 +198619.774}
SPL {X  -159.990, Y  +445.900, Z    +0.000, E1   +66.225, E3 +198631.087}
ENDSPLINE

SPLINE
SPL {X  -159.990, Y  +465.730, Z    +0.000, E1   +61.693, E3 +198644.912}
ENDSPLINE

SPLINE
SPL {X  -159.990, Y  +452.456, Z    +0.000, E1   +62.114, E3 +198656.839}
SPL {X  -159.990, Y  +436.367, Z    +0.000, E1   +62.893, E3 +198669.099}
SPL {X  -159.990, Y  +416.857, Z    +0.000, E1   +63.835, E3 +198682.838}
SPL {X  -159.990, Y  +402.942, Z    +0.000, E1   +64.377, E3 +198693.067}
SPL {X  -159.990, Y  +382.745, Z    +0.000, E1   +65.209, E3 +198706.981}
SPL {X  -158.334, Y  +359.539, Z    +0.000, E1   +66.148, E3 +198721.754}
ENDSPLINE

SPLINE
SPL {X  -159.548, Y  +370.618, Z    +0.000, E1   +63.072, E3 +198733.561}
ENDSPLINE

SPLINE
SPL {X  -158.758, Y  +362.683, Z    +0.000, E1   +62.956, E3 +198742.944}
SPL {X  -157.125, Y  +352.357, Z    +0.000, E1   +62.751, E3 +198755.677}
SPL {X  -154.421, Y  +340.656, Z    +0.000, E1   +62.344, E3 +198771.031}
SPL {X  -151.938, Y  +332.383, Z    +0.000, E1   +61.927, E3 +198782.503}
SPL {X  -149.604, Y  +325.796, Z    +0.000, E1   +61.568, E3 +198791.889}
SPL {X  -147.413, Y  +320.320, Z    +0.000, E1   +61.198, E3 +198799.942}
SPL {X  -145.235, Y  +315.391, Z    +0.000, E1   +60.847, E3 +198807.317}
SPL {X  -141.610, Y  +308.046, Z    +0.000, E1   +60.266, E3 +198818.553}
SPL {X  -138.010, Y  +301.568, Z    +0.000, E1   +59.585, E3 +198828.825}
SPL {X  -134.884, Y  +296.459, Z    +0.000, E1   +59.021, E3 +198837.006}
SPL {X  -132.471, Y  +292.789, Z    +0.000, E1   +58.532, E3 +198842.998}
SPL {X  -113.391, Y  +269.632, Z    +0.000, E1   +50.631, E3 +198938.046}
ENDSPLINE

SPLINE
SPL {X  -117.172, Y  +273.562, Z    +0.000, E1   +47.526, E3 +198986.197}
SPL {X  -141.985, Y  +308.763, Z    +0.000, E1   +38.695, E3 +199053.507}
SPL {X  -151.595, Y  +331.355, Z    +0.000, E1   +30.702, E3 +199068.026}
SPL {X  -155.358, Y  +344.279, Z    +0.000, E1   +24.937, E3 +199073.214}
SPL {X  -158.582, Y  +361.322, Z    +0.000, E1   +15.773, E3 +199077.558}
SPL {X  -159.657, Y  +372.183, Z    +0.000, E1    +8.995, E3 +199079.166}
SPL {X  -159.949, Y  +378.873, Z    +0.000, E1    +4.398, E3 +199079.740}
SPL {X  -159.990, Y  +382.801, Z    +0.000, E1    +1.461, E3 +199079.914}
SPL {X  -159.990, Y  +385.055, Z    +0.000, E1    -0.429, E3 +199079.953}
SPL {X  -159.990, Y  +388.743, Z    +0.000, E1    -5.147, E3 +199080.094}
SPL {X  -159.990, Y  +394.848, Z    +0.000, E1   -14.441, E3 +199080.634}
SPL {X  -159.990, Y  +402.771, Z    +0.000, E1   -27.045, E3 +199081.886}
SPL {X  -159.990, Y  +416.096, Z    +0.000, E1   -42.325, E3 +199085.554}
SPL {X  -159.990, Y  +469.763, Z    +0.000, E1   -60.937, E3 +199110.783}
SPL {X  -159.990, Y  +561.242, Z    +0.000, E1   -63.988, E3 +199181.732}
SPL {X  -159.990, Y  +574.019, Z    +0.000, E1   -64.020, E3 +199194.898}
SPL {X  -159.990, Y  +591.720, Z    +0.000, E1   -64.032, E3 +199213.196}
SPL {X  -159.990, Y  +605.088, Z    +0.000, E1   -63.988, E3 +199227.124}
SPL {X  -159.990, Y  +614.683, Z    +0.000, E1   -63.997, E3 +199237.018}
SPL {X  -159.990, Y  +629.274, Z    +0.000, E1   -64.033, E3 +199252.049}
SPL {X  -159.990, Y  +645.396, Z    +0.000, E1   -64.010, E3 +199268.780}
SPL {X  -159.990, Y  +656.294, Z    +0.000, E1   -63.988, E3 +199280.110}
SPL {X  -159.990, Y  +667.666, Z    +0.000, E1   -64.016, E3 +199291.802}
SPL {X  -159.767, Y  +679.937, Z    +0.000, E1   -63.968, E3 +199304.777}
SPL {X  -159.113, Y  +688.225, Z    +0.000, E1   -63.867, E3 +199314.055}
SPL {X  -158.361, Y  +694.273, Z    +0.000, E1   -63.762, E3 +199321.092}
SPL {X  -157.131, Y  +701.612, Z    +0.000, E1   -63.591, E3 +199329.965}
SPL {X  -154.918, Y  +711.464, Z    +0.000, E1   -63.294, E3 +199342.401}
SPL {X  -151.874, Y  +721.810, Z    +0.000, E1   -62.834, E3 +199356.207}
SPL {X  -148.087, Y  +732.056, Z    +0.000, E1   -62.252, E3 +199370.564}
SPL {X  -144.667, Y  +739.825, Z    +0.000, E1   -61.658, E3 +199381.953}
SPL {X  -142.263, Y  +744.698, Z    +0.000, E1   -61.245, E3 +199389.269}
SPL {X  -138.935, Y  +750.833, Z    +0.000, E1   -60.711, E3 +199398.593}
SPL {X  -135.668, Y  +756.300, Z    +0.000, E1   -60.086, E3 +199407.156}
SPL {X  -132.995, Y  +760.433, Z    +0.000, E1   -59.601, E3 +199413.664}
SPL {X  -109.949, Y  +787.724, Z    +0.000, E1   -51.944, E3 +199506.226}
ENDSPLINE

SPLINE
SPL {X  -129.366, Y  +765.635, Z    +0.000, E1   -44.361, E3 +199615.968}
SPL {X  -144.719, Y  +739.715, Z    +0.000, E1   -37.620, E3 +199642.815}
SPL {X  -154.606, Y  +712.654, Z    +0.000, E1   -26.872, E3 +199656.035}
SPL {X  -158.229, Y  +695.175, Z    +0.000, E1   -17.621, E3 +199660.521}
SPL {X  -159.735, Y  +680.532, Z    +0.000, E1    -8.352, E3 +199662.613}
SPL {X  -159.976, Y  +673.579, Z    +0.000, E1    -3.308, E3 +199663.108}
SPL {X  -159.990, Y  +669.438, Z    +0.000, E1    -0.061, E3 +199663.205}
SPL {X  -159.990, Y  +667.221, Z    +0.000, E1    +2.789, E3 +199663.248}
SPL {X  -159.990, Y  +663.611, Z    +0.000, E1    +7.967, E3 +199663.439}
SPL {X  -159.990, Y  +658.381, Z    +0.000, E1   +16.786, E3 +199663.919}
SPL {X  -159.990, Y  +651.878, Z    +0.000, E1   +27.298, E3 +199664.918}
SPL {X  -159.990, Y  +644.587, Z    +0.000, E1   +37.284, E3 +199666.501}
SPL {X  -159.990, Y  +633.621, Z    +0.000, E1   +47.309, E3 +199669.992}
SPL {X  -159.990, Y  +588.658, Z    +0.000, E1   +60.812, E3 +199692.312}
SPL {X  -159.990, Y  +495.038, Z    +0.000, E1   +63.580, E3 +199767.548}
SPL {X  -159.990, Y  +483.848, Z    +0.000, E1   +63.590, E3 +199779.333}
SPL {X  -159.990, Y  +471.874, Z    +0.000, E1   +63.586, E3 +199791.959}
SPL {X  -159.990, Y  +461.079, Z    +0.000, E1   +63.579, E3 +199803.367}
SPL {X  -159.990, Y  +450.188, Z    +0.000, E1   +63.581, E3 +199814.858}
SPL {X  -159.990, Y  +442.553, Z    +0.000, E1   +63.337, E3 +199824.682}
ENDSPLINE

SPLINE
SPL {X  -159.990, Y  +465.419, Z    +0.000, E1   +58.181, E3 +199833.527}
ENDSPLINE

SPLINE
SPL {X  -159.990, Y  +455.003, Z    +0.000, E1   +58.788, E3 +199843.065}
SPL {X  -159.990, Y  +443.180, Z    +0.000, E1   +59.522, E3 +199853.103}
SPL {X  -159.990, Y  +431.227, Z    +0.000, E1   +60.120, E3 +199863.796}
SPL {X  -159.990, Y  +413.464, Z    +0.000, E1   +61.043, E3 +199878.786}
SPL {X  -159.990, Y  +395.417, Z    +0.000, E1   +62.063, E3 +199892.228}
SPL {X  -159.983, Y  +381.042, Z    +0.000, E1   +62.802, E3 +199902.860}
SPL {X  -159.542, Y  +370.537, Z    +0.000, E1   +63.069, E3 +199912.242}
SPL {X  -158.758, Y  +362.683, Z    +0.000, E1   +62.956, E3 +199921.515}
SPL {X  -157.125, Y  +352.357, Z    +0.000, E1   +62.751, E3 +199934.249}
SPL {X  -154.421, Y  +340.656, Z    +0.000, E1   +62.344, E3 +199949.602}
SPL {X  -151.938, Y  +332.383, Z    +0.000, E1   +61.927, E3 +199961.075}
SPL {X  -149.604, Y  +325.796, Z    +0.000, E1   +61.568, E3 +199970.461}
SPL {X  -147.413, Y  +320.320, Z    +0.000, E1   +61.198, E3 +199978.514}
SPL {X  -145.235, Y  +315.391, Z    +0.000, E1   +60.847, E3 +199985.888}
SPL {X  -141.610, Y  +308.046, Z    +0.000, E1   +60.266, E3 +199997.125}
SPL {X  -138.010, Y  +301.568, Z    +0.000, E1   +59.585, E3 +200007.396}
SPL {X  -134.495, Y  +295.853, Z    +0.000, E1   +58.965, E3 +200016.533}
SPL {X  -113.541, Y  +269.782, Z    +0.000, E1   +50.113, E3 +200124.126}
ENDSPLINE

SPLINE
SPL {X  -141.985, Y  +308.763, Z    +0.000, E1   +38.695, E3 +200232.078}
SPL {X  -154.491, Y  +340.913, Z    +0.000, E1   +26.570, E3 +200250.531}
SPL {X  -158.582, Y  +361.322, Z    +0.000, E1   +15.773, E3 +200256.129}
SPL {X  -159.657, Y  +372.183, Z    +0.000, E1    +8.995, E3 +200257.738}
SPL {X  -159.949, Y  +378.873, Z    +0.000, E1    +4.398, E3 +200258.312}
SPL {X  -159.990, Y  +384.063, Z    +0.000, E1    +0.515, E3 +200258.508}
SPL {X  -159.990, Y  +386.497, Z    +0.000, E1    -2.123, E3 +200258.564}
SPL {X  -159.990, Y  +391.572, Z    +0.000, E1    -9.236, E3 +200258.870}
SPL {X  -159.990, Y  +397.198, Z    +0.000, E1   -18.490, E3 +200259.494}
SPL {X  -159.990, Y  +402.771, Z    +0.000, E1   -27.045, E3 +200260.458}
SPL {X  -159.990, Y  +416.096, Z    +0.000, E1   -42.325, E3 +200264.125}
SPL {X  -159.990, Y  +469.763, Z    +0.000, E1   -60.937, E3 +200289.355}
SPL {X  -159.990, Y  +565.969, Z    +0.000, E1   -64.023, E3 +200365.129}
SPL {X  -159.990, Y  +578.082, Z    +0.000, E1   -63.987, E3 +200377.737}
SPL {X  -159.990, Y  +588.139, Z    +0.000, E1   -64.000, E3 +200388.117}
SPL {X  -159.990, Y  +601.786, Z    +0.000, E1   -64.016, E3 +200402.221}
SPL {X  -159.990, Y  +618.770, Z    +0.000, E1   -64.031, E3 +200419.757}
SPL {X  -159.990, Y  +632.928, Z    +0.000, E1   -63.998, E3 +200434.466}
SPL {X  -159.990, Y  +645.396, Z    +0.000, E1   -64.010, E3 +200447.352}
SPL {X  -159.990, Y  +659.675, Z    +0.000, E1   -64.013, E3 +200462.124}
SPL {X  -159.990, Y  +670.719, Z    +0.000, E1   -63.993, E3 +200473.573}
SPL {X  -159.767, Y  +679.937, Z    +0.000, E1   -63.968, E3 +200483.348}
SPL {X  -158.736, Y  +691.491, Z    +0.000, E1   -63.843, E3 +200496.347}
SPL {X  -157.131, Y  +701.612, Z    +0.000, E1   -63.591, E3 +200508.537}
SPL {X  -155.594, Y  +708.746, Z    +0.000, E1   -63.361, E3 +200517.517}
SPL {X  -153.286, Y  +717.329, Z    +0.000, E1   -63.046, E3 +200528.725}
SPL {X  -150.953, Y  +724.510, Z    +0.000, E1   -62.654, E3 +200538.553}
SPL {X  -148.087, Y  +732.056, Z    +0.000, E1   -62.252, E3 +200549.135}
SPL {X  -144.667, Y  +739.825, Z    +0.000, E1   -61.658, E3 +200560.525}
SPL {X  -142.263, Y  +744.698, Z    +0.000, E1   -61.245, E3 +200567.840}
SPL {X  -139.956, Y  +749.019, Z    +0.000, E1   -60.852, E3 +200574.418}
SPL {X  -136.617, Y  +754.762, Z    +0.000, E1   -60.296, E3 +200583.272}
SPL {X  -132.995, Y  +760.433, Z    +0.000, E1   -59.601, E3 +200592.235}
SPL {X  -109.949, Y  +787.724, Z    +0.000, E1   -51.944, E3 +200684.797}
ENDSPLINE

SPLINE
SPL {X  -129.366, Y  +765.635, Z    +0.000, E1   -44.361, E3 +200794.539}
SPL {X  -144.719, Y  +739.715, Z    +0.000, E1   -37.620, E3 +200821.386}
SPL {X  -154.606, Y  +712.654, Z    +0.000, E1   -26.872, E3 +200834.606}
SPL {X  -158.229, Y  +695.175, Z    +0.000, E1   -17.621, E3 +200839.092}
SPL {X  -159.536, Y  +683.548, Z    +0.000, E1   -10.326, E3 +200840.880}
SPL {X  -159.946, Y  +675.243, Z    +0.000, E1    -4.608, E3 +200841.589}
SPL {X  -159.990, Y  +669.438, Z    +0.000, E1    -0.061, E3 +200841.777}
SPL {X  -159.990, Y  +666.135, Z    +0.000, E1    +4.178, E3 +200841.868}
SPL {X  -159.990, Y  +662.249, Z    +0.000, E1   +10.338, E3 +200842.099}
SPL {X  -159.990, Y  +658.381, Z    +0.000, E1   +16.786, E3 +200842.491}
SPL {X  -159.990, Y  +651.878, Z    +0.000, E1   +27.298, E3 +200843.490}
SPL {X  -159.990, Y  +644.587, Z    +0.000, E1   +37.284, E3 +200845.073}
SPL {X  -159.990, Y  +633.621, Z    +0.000, E1   +47.309, E3 +200848.564}
SPL {X  -159.990, Y  +588.658, Z    +0.000, E1   +60.812, E3 +200870.884}
SPL {X  -159.990, Y  +495.038, Z    +0.000, E1   +63.580, E3 +200946.120}
SPL {X  -159.990, Y  +483.848, Z    +0.000, E1   +63.590, E3 +200957.905}
SPL {X  -159.990, Y  +471.874, Z    +0.000, E1   +63.586, E3 +200970.530}
SPL {X  -159.990, Y  +461.079, Z    +0.000, E1   +63.579, E3 +200981.939}
SPL {X  -159.990, Y  +450.188, Z    +0.000, E1   +63.581, E3 +200993.429}
SPL {X  -159.990, Y  +442.553, Z    +0.000, E1   +63.337, E3 +201003.253}
ENDSPLINE

SPLINE
SPL {X  -159.990, Y  +465.419, Z    +0.000, E1   +58.181, E3 +201012.098}
ENDSPLINE

SPLINE
SPL {X  -159.990, Y  +455.003, Z    +0.000, E1   +58.788, E3 +201021.637}
SPL {X  -159.990, Y  +443.180, Z    +0.000, E1   +59.522, E3 +201031.675}
SPL {X  -159.990, Y  +431.227, Z    +0.000, E1   +60.120, E3 +201042.367}
SPL {X  -159.990, Y  +418.989, Z    +0.000, E1   +60.714, E3 +201053.002}
SPL {X  -159.990, Y  +401.382, Z    +0.000, E1   +61.735, E3 +201066.471}
SPL {X  -159.983, Y  +381.042, Z    +0.000, E1   +62.802, E3 +201081.431}
SPL {X  -159.542, Y  +370.537, Z    +0.000, E1   +63.069, E3 +201090.813}
SPL {X  -158.287, Y  +359.218, Z    +0.000, E1   +62.927, E3 +201104.228}
SPL {X  -155.813, Y  +346.180, Z    +0.000, E1   +62.560, E3 +201120.805}
SPL {X  -152.656, Y  +334.615, Z    +0.000, E1   +62.078, E3 +201136.457}
SPL {X  -149.604, Y  +325.796, Z    +0.000, E1   +61.568, E3 +201149.032}
SPL {X  -147.413, Y  +320.320, Z    +0.000, E1   +61.198, E3 +201157.085}
SPL {X  -145.235, Y  +315.391, Z    +0.000, E1   +60.847, E3 +201164.460}
SPL {X  -141.610, Y  +308.046, Z    +0.000, E1   +60.266, E3 +201175.696}
SPL {X  -138.010, Y  +301.568, Z    +0.000, E1   +59.585, E3 +201185.967}
SPL {X  -134.884, Y  +296.459, Z    +0.000, E1   +59.021, E3 +201194.149}
SPL {X  -132.471, Y  +292.789, Z    +0.000, E1   +58.532, E3 +201200.140}
SPL {X  -113.391, Y  +269.632, Z    +0.000, E1   +50.631, E3 +201295.188}
ENDSPLINE

SPLINE
SPL {X  -117.172, Y  +273.562, Z    +0.000, E1   +47.526, E3 +201343.340}
SPL {X  -141.985, Y  +308.763, Z    +0.000, E1   +38.695, E3 +201410.650}
SPL {X  -151.595, Y  +331.355, Z    +0.000, E1   +30.702, E3 +201425.169}
SPL {X  -155.358, Y  +344.279, Z    +0.000, E1   +24.937, E3 +201430.357}
SPL {X  -158.582, Y  +361.322, Z    +0.000, E1   +15.773, E3 +201434.701}
SPL {X  -159.657, Y  +372.183, Z    +0.000, E1    +8.995, E3 +201436.309}
SPL {X  -159.949, Y  +378.873, Z    +0.000, E1    +4.398, E3 +201436.883}
SPL {X  -159.990, Y  +382.801, Z    +0.000, E1    +1.461, E3 +201437.057}
SPL {X  -159.990, Y  +385.055, Z    +0.000, E1    -0.429, E3 +201437.096}
SPL {X  -159.990, Y  +388.743, Z    +0.000, E1    -5.147, E3 +201437.237}
SPL {X  -159.990, Y  +394.848, Z    +0.000, E1   -14.441, E3 +201437.777}
SPL {X  -159.990, Y  +402.771, Z    +0.000, E1   -27.045, E3 +201439.029}
SPL {X  -159.990, Y  +416.096, Z    +0.000, E1   -42.325, E3 +201442.696}
SPL {X  -159.990, Y  +469.763, Z    +0.000, E1   -60.937, E3 +201467.926}
SPL {X  -159.990, Y  +565.969, Z    +0.000, E1   -64.023, E3 +201543.700}
SPL {X  -159.990, Y  +578.082, Z    +0.000, E1   -63.987, E3 +201556.309}
SPL {X  -159.990, Y  +591.720, Z    +0.000, E1   -64.032, E3 +201570.339}
SPL {X  -159.990, Y  +605.088, Z    +0.000, E1   -63.988, E3 +201584.266}
SPL {X  -159.990, Y  +618.770, Z    +0.000, E1   -64.031, E3 +201598.329}
SPL {X  -159.990, Y  +632.928, Z    +0.000, E1   -63.998, E3 +201613.037}
SPL {X  -159.990, Y  +645.396, Z    +0.000, E1   -64.010, E3 +201625.923}
SPL {X  -159.990, Y  +659.675, Z    +0.000, E1   -64.013, E3 +201640.695}
SPL {X  -159.990, Y  +670.719, Z    +0.000, E1   -63.993, E3 +201652.145}
SPL {X  -159.767, Y  +679.937, Z    +0.000, E1   -63.968, E3 +201661.920}
SPL {X  -159.113, Y  +688.225, Z    +0.000, E1   -63.867, E3 +201671.198}
SPL {X  -158.361, Y  +694.273, Z    +0.000, E1   -63.762, E3 +201678.235}
SPL {X  -157.131, Y  +701.612, Z    +0.000, E1   -63.591, E3 +201687.108}
SPL {X  -155.594, Y  +708.746, Z    +0.000, E1   -63.361, E3 +201696.088}
SPL {X  -153.286, Y  +717.329, Z    +0.000, E1   -63.046, E3 +201707.297}
SPL {X  -150.233, Y  +726.516, Z    +0.000, E1   -62.565, E3 +201719.890}
SPL {X  -147.385, Y  +733.745, Z    +0.000, E1   -62.104, E3 +201730.194}
SPL {X  -144.667, Y  +739.825, Z    +0.000, E1   -61.658, E3 +201739.096}
SPL {X  -142.263, Y  +744.698, Z    +0.000, E1   -61.245, E3 +201746.412}
SPL {X  -138.935, Y  +750.833, Z    +0.000, E1   -60.711, E3 +201755.736}
SPL {X  -135.668, Y  +756.300, Z    +0.000, E1   -60.086, E3 +201764.299}
SPL {X  -132.995, Y  +760.433, Z    +0.000, E1   -59.601, E3 +201770.807}
SPL {X  -109.949, Y  +787.724, Z    +0.000, E1   -51.944, E3 +201863.368}
ENDSPLINE

SPLINE
SPL {X  -129.366, Y  +765.635, Z    +0.000, E1   -44.361, E3 +201973.110}
SPL {X  -144.719, Y  +739.715, Z    +0.000, E1   -37.620, E3 +201999.958}
SPL {X  -154.606, Y  +712.654, Z    +0.000, E1   -26.872, E3 +202013.178}
SPL {X  -158.229, Y  +695.175, Z    +0.000, E1   -17.621, E3 +202017.664}
SPL {X  -159.536, Y  +683.548, Z    +0.000, E1   -10.326, E3 +202019.452}
SPL {X  -159.946, Y  +675.243, Z    +0.000, E1    -4.608, E3 +202020.160}
SPL {X  -159.990, Y  +670.644, Z    +0.000, E1    -1.007, E3 +202020.335}
SPL {X  -159.990, Y  +668.624, Z    +0.000, E1    +0.752, E3 +202020.362}
SPL {X  -159.990, Y  +663.611, Z    +0.000, E1    +7.967, E3 +202020.582}
SPL {X  -159.990, Y  +658.381, Z    +0.000, E1   +16.786, E3 +202021.062}
SPL {X  -159.990, Y  +651.878, Z    +0.000, E1   +27.298, E3 +202022.061}
SPL {X  -159.990, Y  +644.587, Z    +0.000, E1   +37.284, E3 +202023.644}
SPL {X  -159.990, Y  +633.621, Z    +0.000, E1   +47.309, E3 +202027.135}
SPL {X  -159.990, Y  +588.658, Z    +0.000, E1   +60.812, E3 +202049.455}
SPL {X  -159.990, Y  +495.038, Z    +0.000, E1   +63.580, E3 +202124.691}
SPL {X  -159.990, Y  +483.848, Z    +0.000, E1   +63.590, E3 +202136.476}
SPL {X  -159.990, Y  +471.874, Z    +0.000, E1   +63.586, E3 +202149.102}
SPL {X  -159.990, Y  +461.079, Z    +0.000, E1   +63.579, E3 +202160.510}
SPL {X  -159.990, Y  +450.188, Z    +0.000, E1   +63.581, E3 +202172.001}
SPL {X  -159.990, Y  +442.553, Z    +0.000, E1   +63.337, E3 +202181.824}
ENDSPLINE

SPLINE
SPL {X  -159.990, Y  +465.419, Z    +0.000, E1   +58.181, E3 +202190.670}
ENDSPLINE

SPLINE
SPL {X  -159.990, Y  +455.003, Z    +0.000, E1   +58.788, E3 +202200.208}
SPL {X  -159.990, Y  +443.180, Z    +0.000, E1   +59.522, E3 +202210.246}
SPL {X  -159.990, Y  +431.227, Z    +0.000, E1   +60.120, E3 +202220.938}
SPL {X  -159.990, Y  +418.989, Z    +0.000, E1   +60.714, E3 +202231.574}
SPL {X  -159.990, Y  +401.382, Z    +0.000, E1   +61.735, E3 +202245.043}
SPL {X  -159.983, Y  +381.042, Z    +0.000, E1   +62.802, E3 +202260.003}
SPL {X  -159.542, Y  +370.537, Z    +0.000, E1   +63.069, E3 +202269.385}
SPL {X  -158.758, Y  +362.683, Z    +0.000, E1   +62.956, E3 +202278.658}
SPL {X  -157.125, Y  +352.357, Z    +0.000, E1   +62.751, E3 +202291.392}
SPL {X  -154.421, Y  +340.656, Z    +0.000, E1   +62.344, E3 +202306.745}
SPL {X  -151.938, Y  +332.383, Z    +0.000, E1   +61.927, E3 +202318.218}
SPL {X  -149.604, Y  +325.796, Z    +0.000, E1   +61.568, E3 +202327.603}
SPL {X  -147.413, Y  +320.320, Z    +0.000, E1   +61.198, E3 +202335.657}
SPL {X  -145.235, Y  +315.391, Z    +0.000, E1   +60.847, E3 +202343.031}
SPL {X  -142.998, Y  +310.747, Z    +0.000, E1   +60.455, E3 +202350.144}
SPL {X  -140.747, Y  +306.427, Z    +0.000, E1   +60.074, E3 +202356.853}
SPL {X  -138.010, Y  +301.568, Z    +0.000, E1   +59.585, E3 +202364.539}
SPL {X  -134.495, Y  +295.853, Z    +0.000, E1   +58.965, E3 +202373.676}
SPL {X  -113.391, Y  +269.632, Z    +0.000, E1   +50.631, E3 +202473.760}
ENDSPLINE

SPLINE
SPL {X  -117.172, Y  +273.562, Z    +0.000, E1   +47.526, E3 +202521.911}
SPL {X  -141.985, Y  +308.763, Z    +0.000, E1   +38.695, E3 +202589.221}
SPL {X  -151.595, Y  +331.355, Z    +0.000, E1   +30.702, E3 +202603.740}
SPL {X  -155.358, Y  +344.279, Z    +0.000, E1   +24.937, E3 +202608.929}
SPL {X  -158.582, Y  +361.322, Z    +0.000, E1   +15.773, E3 +202613.272}
SPL {X  -159.657, Y  +372.183, Z    +0.000, E1    +8.995, E3 +202614.880}
SPL {X  -159.949, Y  +378.873, Z    +0.000, E1    +4.398, E3 +202615.455}
SPL {X  -159.990, Y  +382.801, Z    +0.000, E1    +1.461, E3 +202615.628}
SPL {X  -159.990, Y  +385.055, Z    +0.000, E1    -0.429, E3 +202615.668}
SPL {X  -159.990, Y  +388.743, Z    +0.000, E1    -5.147, E3 +202615.808}
SPL {X  -159.990, Y  +393.154, Z    +0.000, E1   -11.942, E3 +202616.140}
SPL {X  -159.990, Y  +397.198, Z    +0.000, E1   -18.490, E3 +202616.637}
SPL {X  -159.990, Y  +402.771, Z    +0.000, E1   -27.045, E3 +202617.601}
SPL {X  -159.990, Y  +416.096, Z    +0.000, E1   -42.325, E3 +202621.268}
SPL {X  -159.990, Y  +469.763, Z    +0.000, E1   -60.937, E3 +202646.498}
SPL {X  -159.990, Y  +565.969, Z    +0.000, E1   -64.023, E3 +202722.272}
SPL {X  -159.990, Y  +578.082, Z    +0.000, E1   -63.987, E3 +202734.880}
SPL {X  -159.990, Y  +588.139, Z    +0.000, E1   -64.000, E3 +202745.260}
SPL {X  -159.990, Y  +601.786, Z    +0.000, E1   -64.016, E3 +202759.364}
SPL {X  -159.990, Y  +618.770, Z    +0.000, E1   -64.031, E3 +202776.900}
SPL {X  -159.990, Y  +636.111, Z    +0.000, E1   -64.024, E3 +202794.855}
SPL {X  -159.990, Y  +648.153, Z    +0.000, E1   -63.990, E3 +202807.387}
SPL {X  -159.990, Y  +659.675, Z    +0.000, E1   -64.013, E3 +202819.267}
SPL {X  -159.990, Y  +670.719, Z    +0.000, E1   -63.993, E3 +202830.716}
SPL {X  -159.767, Y  +679.937, Z    +0.000, E1   -63.968, E3 +202840.491}
SPL {X  -158.736, Y  +691.491, Z    +0.000, E1   -63.843, E3 +202853.490}
SPL {X  -157.131, Y  +701.612, Z    +0.000, E1   -63.591, E3 +202865.680}
SPL {X  -155.594, Y  +708.746, Z    +0.000, E1   -63.361, E3 +202874.660}
SPL {X  -153.286, Y  +717.329, Z    +0.000, E1   -63.046, E3 +202885.868}
SPL {X  -150.233, Y  +726.516, Z    +0.000, E1   -62.565, E3 +202898.461}
SPL {X  -147.385, Y  +733.745, Z    +0.000, E1   -62.104, E3 +202908.766}
SPL {X  -144.667, Y  +739.825, Z    +0.000, E1   -61.658, E3 +202917.668}
SPL {X  -142.263, Y  +744.698, Z    +0.000, E1   -61.245, E3 +202924.983}
SPL {X  -138.935, Y  +750.833, Z    +0.000, E1   -60.711, E3 +202934.307}
SPL {X  -135.668, Y  +756.300, Z    +0.000, E1   -60.086, E3 +202942.871}
SPL {X  -132.995, Y  +760.433, Z    +0.000, E1   -59.601, E3 +202949.378}
SPL {X  -109.949, Y  +787.724, Z    +0.000, E1   -51.944, E3 +203041.940}
ENDSPLINE

SPLINE
SPL {X  -129.366, Y  +765.635, Z    +0.000, E1   -44.361, E3 +203151.682}
SPL {X  -144.719, Y  +739.715, Z    +0.000, E1   -37.620, E3 +203178.529}
SPL {X  -154.606, Y  +712.654, Z    +0.000, E1   -26.872, E3 +203191.749}
SPL {X  -158.229, Y  +695.175, Z    +0.000, E1   -17.621, E3 +203196.235}
SPL {X  -159.735, Y  +680.532, Z    +0.000, E1    -8.352, E3 +203198.328}
SPL {X  -159.990, Y  +671.731, Z    +0.000, E1    -1.953, E3 +203198.877}
SPL {X  -159.990, Y  +669.188, Z    +0.000, E1    +0.261, E3 +203198.922}
SPL {X  -159.990, Y  +666.135, Z    +0.000, E1    +4.178, E3 +203199.011}
SPL {X  -159.990, Y  +662.249, Z    +0.000, E1   +10.338, E3 +203199.242}
SPL {X  -159.990, Y  +658.381, Z    +0.000, E1   +16.786, E3 +203199.634}
SPL {X  -159.990, Y  +651.878, Z    +0.000, E1   +27.298, E3 +203200.633}
SPL {X  -159.990, Y  +644.587, Z    +0.000, E1   +37.284, E3 +203202.216}
SPL {X  -159.990, Y  +633.621, Z    +0.000, E1   +47.309, E3 +203205.707}
SPL {X  -159.990, Y  +588.658, Z    +0.000, E1   +60.812, E3 +203228.026}
SPL {X  -159.990, Y  +495.038, Z    +0.000, E1   +63.580, E3 +203303.263}
SPL {X  -159.990, Y  +483.848, Z    +0.000, E1   +63.590, E3 +203315.047}
SPL {X  -159.990, Y  +471.874, Z    +0.000, E1   +63.586, E3 +203327.673}
SPL {X  -159.990, Y  +461.079, Z    +0.000, E1   +63.579, E3 +203339.082}
SPL {X  -159.990, Y  +450.188, Z    +0.000, E1   +63.581, E3 +203350.572}
SPL {X  -159.990, Y  +442.553, Z    +0.000, E1   +63.337, E3 +203360.396}
ENDSPLINE

SPLINE
SPL {X  -159.990, Y  +465.419, Z    +0.000, E1   +58.181, E3 +203369.241}
ENDSPLINE

SPLINE
SPL {X  -159.990, Y  +455.003, Z    +0.000, E1   +58.788, E3 +203378.779}
SPL {X  -159.990, Y  +443.180, Z    +0.000, E1   +59.522, E3 +203388.818}
SPL {X  -159.990, Y  +431.227, Z    +0.000, E1   +60.120, E3 +203399.510}
SPL {X  -159.990, Y  +413.464, Z    +0.000, E1   +61.043, E3 +203414.500}
SPL {X  -159.990, Y  +395.417, Z    +0.000, E1   +62.063, E3 +203427.943}
SPL {X  -159.983, Y  +381.042, Z    +0.000, E1   +62.802, E3 +203438.574}
SPL {X  -159.542, Y  +370.537, Z    +0.000, E1   +63.069, E3 +203447.956}
SPL {X  -158.287, Y  +359.218, Z    +0.000, E1   +62.927, E3 +203461.371}
SPL {X  -156.553, Y  +349.515, Z    +0.000, E1   +62.627, E3 +203473.682}
SPL {X  -154.421, Y  +340.656, Z    +0.000, E1   +62.344, E3 +203485.316}
SPL {X  -151.938, Y  +332.383, Z    +0.000, E1   +61.927, E3 +203496.789}
SPL {X  -149.604, Y  +325.796, Z    +0.000, E1   +61.568, E3 +203506.175}
SPL {X  -147.413, Y  +320.320, Z    +0.000, E1   +61.198, E3 +203514.228}
SPL {X  -145.235, Y  +315.391, Z    +0.000, E1   +60.847, E3 +203521.603}
SPL {X  -141.610, Y  +308.046, Z    +0.000, E1   +60.266, E3 +203532.839}
SPL {X  -138.010, Y  +301.568, Z    +0.000, E1   +59.585, E3 +203543.110}
SPL {X  -134.495, Y  +295.853, Z    +0.000, E1   +58.965, E3 +203552.248}
SPL {X  -113.541, Y  +269.782, Z    +0.000, E1   +50.113, E3 +203659.840}
ENDSPLINE

SPLINE
SPL {X  -141.985, Y  +308.763, Z    +0.000, E1   +38.695, E3 +203767.793}
SPL {X  -154.491, Y  +340.913, Z    +0.000, E1   +26.570, E3 +203786.245}
SPL {X  -158.582, Y  +361.322, Z    +0.000, E1   +15.773, E3 +203791.844}
SPL {X  -159.657, Y  +372.183, Z    +0.000, E1    +8.995, E3 +203793.452}
SPL {X  -159.949, Y  +378.873, Z    +0.000, E1    +4.398, E3 +203794.026}
SPL {X  -159.990, Y  +384.682, Z    +0.000, E1    +0.050, E3 +203794.233}
SPL {X  -159.990, Y  +388.743, Z    +0.000, E1    -5.147, E3 +203794.380}
SPL {X  -159.990, Y  +394.848, Z    +0.000, E1   -14.441, E3 +203794.920}
SPL {X  -159.990, Y  +402.771, Z    +0.000, E1   -27.045, E3 +203796.172}
SPL {X  -159.990, Y  +414.719, Z    +0.000, E1   -41.161, E3 +203799.346}
SPL {X  -159.990, Y  +424.336, Z    +0.000, E1   -48.481, E3 +203802.781}
SPL {X  -159.990, Y  +469.763, Z    +0.000, E1   -60.937, E3 +203825.069}
SPL {X  -159.990, Y  +561.242, Z    +0.000, E1   -63.988, E3 +203896.017}
SPL {X  -159.990, Y  +574.019, Z    +0.000, E1   -64.020, E3 +203909.184}
SPL {X  -159.990, Y  +591.720, Z    +0.000, E1   -64.032, E3 +203927.482}
SPL {X  -159.990, Y  +605.088, Z    +0.000, E1   -63.988, E3 +203941.409}
SPL {X  -159.990, Y  +614.683, Z    +0.000, E1   -63.997, E3 +203951.304}
SPL {X  -159.990, Y  +629.274, Z    +0.000, E1   -64.033, E3 +203966.335}
SPL {X  -159.990, Y  +645.396, Z    +0.000, E1   -64.010, E3 +203983.066}
SPL {X  -159.990, Y  +656.294, Z    +0.000, E1   -63.988, E3 +203994.396}
SPL {X  -159.990, Y  +667.666, Z    +0.000, E1   -64.016, E3 +204006.087}
SPL {X  -159.767, Y  +679.937, Z    +0.000, E1   -63.968, E3 +204019.063}
SPL {X  -158.736, Y  +691.491, Z    +0.000, E1   -63.843, E3 +204032.061}
SPL {X  -157.131, Y  +701.612, Z    +0.000, E1   -63.591, E3 +204044.251}
SPL {X  -155.594, Y  +708.746, Z    +0.000, E1   -63.361, E3 +204053.231}
SPL {X  -153.286, Y  +717.329, Z    +0.000, E1   -63.046, E3 +204064.440}
SPL {X  -150.953, Y  +724.510, Z    +0.000, E1   -62.654, E3 +204074.268}
SPL {X  -148.087, Y  +732.056, Z    +0.000, E1   -62.252, E3 +204084.850}
SPL {X  -144.667, Y  +739.825, Z    +0.000, E1   -61.658, E3 +204096.239}
SPL {X  -142.263, Y  +744.698, Z    +0.000, E1   -61.245, E3 +204103.554}
SPL {X  -139.956, Y  +749.019, Z    +0.000, E1   -60.852, E3 +204110.132}
SPL {X  -136.617, Y  +754.762, Z    +0.000, E1   -60.296, E3 +204118.986}
SPL {X  -132.995, Y  +760.433, Z    +0.000, E1   -59.601, E3 +204127.950}
SPL {X  -109.949, Y  +787.724, Z    +0.000, E1   -51.944, E3 +204220.511}
ENDSPLINE

SPLINE
SPL {X  -129.366, Y  +765.635, Z    +0.000, E1   -44.361, E3 +204330.253}
SPL {X  -144.719, Y  +739.715, Z    +0.000, E1   -37.620, E3 +204357.101}
SPL {X  -154.606, Y  +712.654, Z    +0.000, E1   -26.872, E3 +204370.321}
SPL {X  -158.229, Y  +695.175, Z    +0.000, E1   -17.621, E3 +204374.807}
SPL {X  -159.735, Y  +680.532, Z    +0.000, E1    -8.352, E3 +204376.899}
SPL {X  -159.990, Y  +671.731, Z    +0.000, E1    -1.953, E3 +204377.449}
SPL {X  -159.990, Y  +669.188, Z    +0.000, E1    +0.261, E3 +204377.493}
SPL {X  -159.990, Y  +666.135, Z    +0.000, E1    +4.178, E3 +204377.582}
SPL {X  -159.990, Y  +662.249, Z    +0.000, E1   +10.338, E3 +204377.813}
SPL {X  -159.990, Y  +658.381, Z    +0.000, E1   +16.786, E3 +204378.205}
SPL {X  -159.990, Y  +651.878, Z    +0.000, E1   +27.298, E3 +204379.204}
SPL {X  -159.990, Y  +644.587, Z    +0.000, E1   +37.284, E3 +204380.787}
SPL {X  -159.990, Y  +633.621, Z    +0.000, E1   +47.309, E3 +204384.278}
SPL {X  -159.990, Y  +588.658, Z    +0.000, E1   +60.812, E3 +204406.598}
SPL {X  -159.990, Y  +495.038, Z    +0.000, E1   +63.580, E3 +204481.834}
SPL {X  -159.990, Y  +483.848, Z    +0.000, E1   +63.590, E3 +204493.619}
SPL {X  -159.990, Y  +471.874, Z    +0.000, E1   +63.586, E3 +204506.245}
SPL {X  -159.990, Y  +461.079, Z    +0.000, E1   +63.579, E3 +204517.653}
SPL {X  -159.990, Y  +450.188, Z    +0.000, E1   +63.581, E3 +204529.144}
SPL {X  -159.990, Y  +442.553, Z    +0.000, E1   +63.337, E3 +204538.967}
ENDSPLINE

SPLINE
SPL {X  -159.990, Y  +465.419, Z    +0.000, E1   +58.181, E3 +204547.813}
ENDSPLINE

SPLINE
SPL {X  -159.990, Y  +455.003, Z    +0.000, E1   +58.788, E3 +204557.351}
SPL {X  -159.990, Y  +443.180, Z    +0.000, E1   +59.522, E3 +204567.389}
SPL {X  -159.990, Y  +431.227, Z    +0.000, E1   +60.120, E3 +204578.081}
SPL {X  -159.990, Y  +413.464, Z    +0.000, E1   +61.043, E3 +204593.071}
SPL {X  -159.990, Y  +395.417, Z    +0.000, E1   +62.063, E3 +204606.514}
SPL {X  -159.983, Y  +381.042, Z    +0.000, E1   +62.802, E3 +204617.145}
SPL {X  -159.542, Y  +370.537, Z    +0.000, E1   +63.069, E3 +204626.527}
SPL {X  -158.758, Y  +362.683, Z    +0.000, E1   +62.956, E3 +204635.801}
SPL {X  -157.125, Y  +352.357, Z    +0.000, E1   +62.751, E3 +204648.534}
SPL {X  -154.421, Y  +340.656, Z    +0.000, E1   +62.344, E3 +204663.888}
SPL {X  -151.938, Y  +332.383, Z    +0.000, E1   +61.927, E3 +204675.360}
SPL {X  -149.604, Y  +325.796, Z    +0.000, E1   +61.568, E3 +204684.746}
SPL {X  -147.413, Y  +320.320, Z    +0.000, E1   +61.198, E3 +204692.799}
SPL {X  -145.235, Y  +315.391, Z    +0.000, E1   +60.847, E3 +204700.174}
SPL {X  -141.610, Y  +308.046, Z    +0.000, E1   +60.266, E3 +204711.410}
SPL {X  -138.010, Y  +301.568, Z    +0.000, E1   +59.585, E3 +204721.682}
SPL {X  -134.495, Y  +295.853, Z    +0.000, E1   +58.965, E3 +204730.819}
SPL {X  -113.541, Y  +269.782, Z    +0.000, E1   +50.113, E3 +204838.412}
ENDSPLINE

SPLINE
SPL {X  -141.985, Y  +308.763, Z    +0.000, E1   +38.695, E3 +204946.364}
SPL {X  -154.491, Y  +340.913, Z    +0.000, E1   +26.570, E3 +204964.816}
SPL {X  -158.582, Y  +361.322, Z    +0.000, E1   +15.773, E3 +204970.415}
SPL {X  -159.657, Y  +372.183, Z    +0.000, E1    +8.995, E3 +204972.023}
SPL {X  -159.949, Y  +378.873, Z    +0.000, E1    +4.398, E3 +204972.598}
SPL {X  -159.990, Y  +384.063, Z    +0.000, E1    +0.515, E3 +204972.794}
SPL {X  -159.990, Y  +386.497, Z    +0.000, E1    -2.123, E3 +204972.850}
SPL {X  -159.990, Y  +389.673, Z    +0.000, E1    -6.604, E3 +204973.003}
SPL {X  -159.990, Y  +394.848, Z    +0.000, E1   -14.441, E3 +204973.491}
SPL {X  -159.990, Y  +402.771, Z    +0.000, E1   -27.045, E3 +204974.743}
SPL {X  -159.990, Y  +414.719, Z    +0.000, E1   -41.161, E3 +204977.918}
SPL {X  -159.990, Y  +424.336, Z    +0.000, E1   -48.481, E3 +204981.352}
SPL {X  -159.990, Y  +469.763, Z    +0.000, E1   -60.937, E3 +205003.641}
SPL {X  -159.990, Y  +561.242, Z    +0.000, E1   -63.988, E3 +205074.589}
SPL {X  -159.990, Y  +574.019, Z    +0.000, E1   -64.020, E3 +205087.755}
SPL {X  -159.990, Y  +588.139, Z    +0.000, E1   -64.000, E3 +205102.403}
SPL {X  -159.990, Y  +601.786, Z    +0.000, E1   -64.016, E3 +205116.507}
SPL {X  -159.990, Y  +614.683, Z    +0.000, E1   -63.997, E3 +205129.875}
SPL {X  -159.990, Y  +629.274, Z    +0.000, E1   -64.033, E3 +205144.906}
SPL {X  -159.990, Y  +645.396, Z    +0.000, E1   -64.010, E3 +205161.637}
SPL {X  -159.990, Y  +656.294, Z    +0.000, E1   -63.988, E3 +205172.967}
SPL {X  -159.990, Y  +667.666, Z    +0.000, E1   -64.016, E3 +205184.659}
SPL {X  -159.767, Y  +679.937, Z    +0.000, E1   -63.968, E3 +205197.634}
SPL {X  -158.736, Y  +691.491, Z    +0.000, E1   -63.843, E3 +205210.633}
SPL {X  -157.131, Y  +701.612, Z    +0.000, E1   -63.591, E3 +205222.823}
SPL {X  -154.918, Y  +711.464, Z    +0.000, E1   -63.294, E3 +205235.258}
SPL {X  -152.656, Y  +719.385, Z    +0.000, E1   -62.921, E3 +205245.826}
SPL {X  -150.233, Y  +726.516, Z    +0.000, E1   -62.565, E3 +205255.604}
SPL {X  -147.385, Y  +733.745, Z    +0.000, E1   -62.104, E3 +205265.908}
SPL {X  -144.667, Y  +739.825, Z    +0.000, E1   -61.658, E3 +205274.811}
SPL {X  -142.263, Y  +744.698, Z    +0.000, E1   -61.245, E3 +205282.126}
SPL {X  -138.935, Y  +750.833, Z    +0.000, E1   -60.711, E3 +205291.450}
SPL {X  -135.668, Y  +756.300, Z    +0.000, E1   -60.086, E3 +205300.014}
SPL {X  -132.995, Y  +760.433, Z    +0.000, E1   -59.601, E3 +205306.521}
SPL {X  -109.949, Y  +787.724, Z    +0.000, E1   -51.944, E3 +205399.083}
ENDSPLINE

SPLINE
SPL {X  -129.366, Y  +765.635, Z    +0.000, E1   -44.361, E3 +205508.825}
SPL {X  -144.719, Y  +739.715, Z    +0.000, E1   -37.620, E3 +205535.672}
SPL {X  -154.606, Y  +712.654, Z    +0.000, E1   -26.872, E3 +205548.892}
SPL {X  -158.229, Y  +695.175, Z    +0.000, E1   -17.621, E3 +205553.378}
SPL {X  -159.735, Y  +680.532, Z    +0.000, E1    -8.352, E3 +205555.470}
SPL {X  -159.976, Y  +673.579, Z    +0.000, E1    -3.308, E3 +205555.965}
SPL {X  -159.990, Y  +669.438, Z    +0.000, E1    -0.061, E3 +205556.062}
SPL {X  -159.990, Y  +666.135, Z    +0.000, E1    +4.178, E3 +205556.154}
SPL {X  -159.990, Y  +662.249, Z    +0.000, E1   +10.338, E3 +205556.385}
SPL {X  -159.990, Y  +658.381, Z    +0.000, E1   +16.786, E3 +205556.777}
SPL {X  -159.990, Y  +651.878, Z    +0.000, E1   +27.298, E3 +205557.776}
SPL {X  -159.990, Y  +644.587, Z    +0.000, E1   +37.284, E3 +205559.358}
SPL {X  -159.990, Y  +633.621, Z    +0.000, E1   +47.309, E3 +205562.849}
SPL {X  -159.990, Y  +588.658, Z    +0.000, E1   +60.812, E3 +205585.169}
SPL {X  -159.990, Y  +495.038, Z    +0.000, E1   +63.580, E3 +205660.406}
SPL {X  -159.990, Y  +483.848, Z    +0.000, E1   +63.590, E3 +205672.190}
SPL {X  -159.990, Y  +471.874, Z    +0.000, E1   +63.586, E3 +205684.816}
SPL {X  -159.990, Y  +461.079, Z    +0.000, E1   +63.579, E3 +205696.225}
SPL {X  -159.990, Y  +450.188, Z    +0.000, E1   +63.581, E3 +205707.715}
SPL {X  -159.990, Y  +442.553, Z    +0.000, E1   +63.337, E3 +205717.539}
ENDSPLINE

SPLINE
SPL {X  -159.990, Y  +465.419, Z    +0.000, E1   +58.181, E3 +205726.384}
ENDSPLINE

SPLINE
SPL {X  -159.990, Y  +455.003, Z    +0.000, E1   +58.788, E3 +205735.922}
SPL {X  -159.990, Y  +443.180, Z    +0.000, E1   +59.522, E3 +205745.961}
SPL {X  -159.990, Y  +431.227, Z    +0.000, E1   +60.120, E3 +205756.653}
SPL {X  -159.990, Y  +413.464, Z    +0.000, E1   +61.043, E3 +205771.643}
SPL {X  -159.990, Y  +395.417, Z    +0.000, E1   +62.063, E3 +205785.086}
SPL {X  -159.983, Y  +381.042, Z    +0.000, E1   +62.802, E3 +205795.717}
SPL {X  -159.542, Y  +370.537, Z    +0.000, E1   +63.069, E3 +205805.099}
SPL {X  -158.287, Y  +359.218, Z    +0.000, E1   +62.927, E3 +205818.514}
SPL {X  -156.553, Y  +349.515, Z    +0.000, E1   +62.627, E3 +205830.825}
SPL {X  -154.421, Y  +340.656, Z    +0.000, E1   +62.344, E3 +205842.459}
SPL {X  -151.938, Y  +332.383, Z    +0.000, E1   +61.927, E3 +205853.932}
SPL {X  -149.604, Y  +325.796, Z    +0.000, E1   +61.568, E3 +205863.318}
SPL {X  -147.413, Y  +320.320, Z    +0.000, E1   +61.198, E3 +205871.371}
SPL {X  -145.235, Y  +315.391, Z    +0.000, E1   +60.847, E3 +205878.746}
SPL {X  -141.610, Y  +308.046, Z    +0.000, E1   +60.266, E3 +205889.982}
SPL {X  -138.010, Y  +301.568, Z    +0.000, E1   +59.585, E3 +205900.253}
SPL {X  -134.495, Y  +295.853, Z    +0.000, E1   +58.965, E3 +205909.391}
SPL {X  -113.541, Y  +269.782, Z    +0.000, E1   +50.113, E3 +206016.983}
ENDSPLINE

SPLINE
SPL {X  -141.985, Y  +308.763, Z    +0.000, E1   +38.695, E3 +206124.935}
SPL {X  -154.491, Y  +340.913, Z    +0.000, E1   +26.570, E3 +206143.388}
SPL {X  -158.582, Y  +361.322, Z    +0.000, E1   +15.773, E3 +206148.987}
SPL {X  -159.657, Y  +372.183, Z    +0.000, E1    +8.995, E3 +206150.595}
SPL {X  -159.949, Y  +378.873, Z    +0.000, E1    +4.398, E3 +206151.169}
SPL {X  -159.990, Y  +384.063, Z    +0.000, E1    +0.515, E3 +206151.365}
SPL {X  -159.990, Y  +386.497, Z    +0.000, E1    -2.123, E3 +206151.421}
SPL {X  -159.990, Y  +391.572, Z    +0.000, E1    -9.236, E3 +206151.727}
SPL {X  -159.990, Y  +397.198, Z    +0.000, E1   -18.490, E3 +206152.352}
SPL {X  -159.990, Y  +402.771, Z    +0.000, E1   -27.045, E3 +206153.315}
SPL {X  -159.990, Y  +416.096, Z    +0.000, E1   -42.325, E3 +206156.982}
SPL {X  -159.990, Y  +469.763, Z    +0.000, E1   -60.937, E3 +206182.212}
SPL {X  -159.990, Y  +565.969, Z    +0.000, E1   -64.023, E3 +206257.986}
SPL {X  -159.990, Y  +578.082, Z    +0.000, E1   -63.987, E3 +206270.594}
SPL {X  -159.990, Y  +588.139, Z    +0.000, E1   -64.000, E3 +206280.975}
SPL {X  -159.990, Y  +601.786, Z    +0.000, E1   -64.016, E3 +206295.078}
SPL {X  -159.990, Y  +618.770, Z    +0.000, E1   -64.031, E3 +206312.615}
SPL {X  -159.990, Y  +636.111, Z    +0.000, E1   -64.024, E3 +206330.569}
SPL {X  -159.990, Y  +652.385, Z    +0.000, E1   -64.020, E3 +206347.427}
SPL {X  -159.990, Y  +667.666, Z    +0.000, E1   -64.016, E3 +206363.230}
SPL {X  -159.767, Y  +679.937, Z    +0.000, E1   -63.968, E3 +206376.206}
SPL {X  -159.113, Y  +688.225, Z    +0.000, E1   -63.867, E3 +206385.483}
SPL {X  -158.361, Y  +694.273, Z    +0.000, E1   -63.762, E3 +206392.521}
SPL {X  -157.131, Y  +701.612, Z    +0.000, E1   -63.591, E3 +206401.394}
SPL {X  -155.594, Y  +708.746, Z    +0.000, E1   -63.361, E3 +206410.374}
SPL {X  -153.286, Y  +717.329, Z    +0.000, E1   -63.046, E3 +206421.582}
SPL {X  -150.233, Y  +726.516, Z    +0.000, E1   -62.565, E3 +206434.176}
SPL {X  -147.385, Y  +733.745, Z    +0.000, E1   -62.104, E3 +206444.480}
SPL {X  -144.667, Y  +739.825, Z    +0.000, E1   -61.658, E3 +206453.382}
SPL {X  -142.263, Y  +744.698, Z    +0.000, E1   -61.245, E3 +206460.697}
SPL {X  -138.935, Y  +750.833, Z    +0.000, E1   -60.711, E3 +206470.022}
SPL {X  -135.668, Y  +756.300, Z    +0.000, E1   -60.086, E3 +206478.585}
SPL {X  -132.995, Y  +760.433, Z    +0.000, E1   -59.601, E3 +206485.093}
SPL {X  -109.949, Y  +787.724, Z    +0.000, E1   -51.944, E3 +206577.654}
ENDSPLINE

SPLINE
SPL {X  -129.366, Y  +765.635, Z    +0.000, E1   -44.361, E3 +206687.396}
SPL {X  -144.719, Y  +739.715, Z    +0.000, E1   -37.620, E3 +206714.244}
SPL {X  -154.606, Y  +712.654, Z    +0.000, E1   -26.872, E3 +206727.464}
SPL {X  -158.229, Y  +695.175, Z    +0.000, E1   -17.621, E3 +206731.950}
SPL {X  -159.536, Y  +683.548, Z    +0.000, E1   -10.326, E3 +206733.737}
SPL {X  -159.946, Y  +675.243, Z    +0.000, E1    -4.608, E3 +206734.446}
SPL {X  -159.990, Y  +670.644, Z    +0.000, E1    -1.007, E3 +206734.621}
SPL {X  -159.990, Y  +669.188, Z    +0.000, E1    +0.261, E3 +206734.636}
SPL {X  -159.990, Y  +666.135, Z    +0.000, E1    +4.178, E3 +206734.725}
SPL {X  -159.990, Y  +662.249, Z    +0.000, E1   +10.338, E3 +206734.956}
SPL {X  -159.990, Y  +658.381, Z    +0.000, E1   +16.786, E3 +206735.348}
SPL {X  -159.990, Y  +651.878, Z    +0.000, E1   +27.298, E3 +206736.347}
SPL {X  -159.990, Y  +644.587, Z    +0.000, E1   +37.284, E3 +206737.930}
SPL {X  -159.990, Y  +633.621, Z    +0.000, E1   +47.309, E3 +206741.421}
SPL {X  -159.990, Y  +588.658, Z    +0.000, E1   +60.812, E3 +206763.741}
SPL {X  -159.990, Y  +495.038, Z    +0.000, E1   +63.580, E3 +206838.977}
SPL {X  -159.990, Y  +483.848, Z    +0.000, E1   +63.590, E3 +206850.762}
SPL {X  -159.990, Y  +471.874, Z    +0.000, E1   +63.586, E3 +206863.387}
SPL {X  -159.990, Y  +461.079, Z    +0.000, E1   +63.579, E3 +206874.796}
SPL {X  -159.990, Y  +450.188, Z    +0.000, E1   +63.581, E3 +206886.287}
SPL {X  -159.990, Y  +442.553, Z    +0.000, E1   +63.337, E3 +206896.110}
ENDSPLINE

SPLINE
SPL {X  -159.990, Y  +465.419, Z    +0.000, E1   +58.181, E3 +206904.956}
ENDSPLINE

SPLINE
SPL {X  -159.990, Y  +455.003, Z    +0.000, E1   +58.788, E3 +206914.494}
SPL {X  -159.990, Y  +443.180, Z    +0.000, E1   +59.522, E3 +206924.532}
SPL {X  -159.990, Y  +431.227, Z    +0.000, E1   +60.120, E3 +206935.224}
SPL {X  -159.990, Y  +418.989, Z    +0.000, E1   +60.714, E3 +206945.859}
SPL {X  -159.990, Y  +401.382, Z    +0.000, E1   +61.735, E3 +206959.329}
SPL {X  -159.983, Y  +381.042, Z    +0.000, E1   +62.802, E3 +206974.288}
SPL {X  -159.542, Y  +370.537, Z    +0.000, E1   +63.069, E3 +206983.670}
SPL {X  -158.758, Y  +362.683, Z    +0.000, E1   +62.956, E3 +206992.944}
SPL {X  -157.125, Y  +352.357, Z    +0.000, E1   +62.751, E3 +207005.677}
SPL {X  -154.421, Y  +340.656, Z    +0.000, E1   +62.344, E3 +207021.031}
SPL {X  -151.938, Y  +332.383, Z    +0.000, E1   +61.927, E3 +207032.503}
SPL {X  -149.604, Y  +325.796, Z    +0.000, E1   +61.568, E3 +207041.889}
SPL {X  -147.413, Y  +320.320, Z    +0.000, E1   +61.198, E3 +207049.942}
SPL {X  -145.235, Y  +315.391, Z    +0.000, E1   +60.847, E3 +207057.317}
SPL {X  -141.610, Y  +308.046, Z    +0.000, E1   +60.266, E3 +207068.553}
SPL {X  -138.010, Y  +301.568, Z    +0.000, E1   +59.585, E3 +207078.825}
SPL {X  -134.495, Y  +295.853, Z    +0.000, E1   +58.965, E3 +207087.962}
SPL {X  -113.541, Y  +269.782, Z    +0.000, E1   +50.113, E3 +207195.554}
ENDSPLINE

SPLINE
SPL {X  -145.506, Y  +315.982, Z    +0.000, E1   +36.457, E3 +207308.790}
SPL {X  -155.358, Y  +344.279, Z    +0.000, E1   +24.937, E3 +207323.214}
SPL {X  -158.582, Y  +361.322, Z    +0.000, E1   +15.773, E3 +207327.558}
SPL {X  -159.657, Y  +372.183, Z    +0.000, E1    +8.995, E3 +207329.166}
SPL {X  -159.986, Y  +381.348, Z    +0.000, E1    +2.678, E3 +207329.855}
SPL {X  -159.990, Y  +384.517, Z    +0.000, E1    +0.022, E3 +207329.944}
SPL {X  -159.990, Y  +385.713, Z    +0.000, E1    -1.275, E3 +207329.965}
SPL {X  -159.990, Y  +388.743, Z    +0.000, E1    -5.147, E3 +207330.094}
SPL {X  -159.990, Y  +393.154, Z    +0.000, E1   -11.942, E3 +207330.426}
SPL {X  -159.990, Y  +397.198, Z    +0.000, E1   -18.490, E3 +207330.923}
SPL {X  -159.990, Y  +402.771, Z    +0.000, E1   -27.045, E3 +207331.886}
SPL {X  -159.990, Y  +416.096, Z    +0.000, E1   -42.325, E3 +207335.554}
SPL {X  -159.990, Y  +469.763, Z    +0.000, E1   -60.937, E3 +207360.783}
SPL {X  -159.990, Y  +561.242, Z    +0.000, E1   -63.988, E3 +207431.732}
SPL {X  -159.990, Y  +574.019, Z    +0.000, E1   -64.020, E3 +207444.898}
SPL {X  -159.990, Y  +591.720, Z    +0.000, E1   -64.032, E3 +207463.196}
SPL {X  -159.990, Y  +605.088, Z    +0.000, E1   -63.988, E3 +207477.124}
SPL {X  -159.990, Y  +614.683, Z    +0.000, E1   -63.997, E3 +207487.018}
SPL {X  -159.990, Y  +629.274, Z    +0.000, E1   -64.033, E3 +207502.049}
SPL {X  -159.990, Y  +645.396, Z    +0.000, E1   -64.010, E3 +207518.780}
SPL {X  -159.990, Y  +656.294, Z    +0.000, E1   -63.988, E3 +207530.110}
SPL {X  -159.990, Y  +667.666, Z    +0.000, E1   -64.016, E3 +207541.802}
SPL {X  -159.767, Y  +679.937, Z    +0.000, E1   -63.968, E3 +207554.777}
SPL {X  -158.736, Y  +691.491, Z    +0.000, E1   -63.843, E3 +207567.775}
SPL {X  -157.131, Y  +701.612, Z    +0.000, E1   -63.591, E3 +207579.965}
SPL {X  -155.594, Y  +708.746, Z    +0.000, E1   -63.361, E3 +207588.946}
SPL {X  -153.286, Y  +717.329, Z    +0.000, E1   -63.046, E3 +207600.154}
SPL {X  -150.953, Y  +724.510, Z    +0.000, E1   -62.654, E3 +207609.982}
SPL {X  -148.087, Y  +732.056, Z    +0.000, E1   -62.252, E3 +207620.564}
SPL {X  -144.667, Y  +739.825, Z    +0.000, E1   -61.658, E3 +207631.953}
SPL {X  -142.263, Y  +744.698, Z    +0.000, E1   -61.245, E3 +207639.269}
SPL {X  -139.956, Y  +749.019, Z    +0.000, E1   -60.852, E3 +207645.846}
SPL {X  -136.617, Y  +754.762, Z    +0.000, E1   -60.296, E3 +207654.700}
SPL {X  -132.995, Y  +760.433, Z    +0.000, E1   -59.601, E3 +207663.664}
SPL {X  -109.949, Y  +787.724, Z    +0.000, E1   -51.944, E3 +207756.226}
ENDSPLINE

